// TIA Portal V17 export
// export: Created 2025-07-01T14:26:13.4361158Z, ExportSetting WithDefaults, DisplayName Totally Integrated Automation Portal, DisplayVersion V17 Update 8, DisplayName TIA Portal Openness, DisplayVersion V17 Update 8, DisplayName TIA Portal Version Control Interface, DisplayVersion V17, DisplayName SINAMICS Startdrive Advanced, DisplayVersion V17 SP2, DisplayName SINAMICS Startdrive G110M, G120, G120C, G120D, G120P, G115D, DisplayVersion V17 SP2, DisplayName SINAMICS Startdrive G130, G150, S120, S150, SINAMICS MV, S210, DisplayVersion V17 SP2, DisplayName STEP 7 Professional, DisplayVersion V17 Update 8, DisplayName SINUMERIK ONE STEP 7 Toolbox, DisplayVersion V17 Update 12, DisplayName SINUMERIK ONE PLC Basic Program Plus, DisplayVersion V17 Update 12, DisplayName SINUMERIK 840D sl STEP 7 Toolbox, DisplayVersion V17 Update 12, DisplayName STEP 7 Safety, DisplayVersion V17 Update 6, DisplayName WinCC Advanced, DisplayVersion V17 Update 8
FUNCTION "FC17100_MAINTENANCE_HMI_SCREEN_VARIABLES" : Void   // FC17100, LAD
{ S7_Optimized_Access := 'TRUE' }
VERSION : 0.1
// stored: AutoNumber false, IsIECCheckEnabled false, SetENOAutomatically false, UDAEnableTagReadback false
   VAR_TEMP
      TEMP : Int;
      NUM_OF_HELPS_TO_0 : Int;
   END_VAR
BEGIN

REGION Network 1: ACTION DONE: POWDER > UNIT 1 > GENERAL
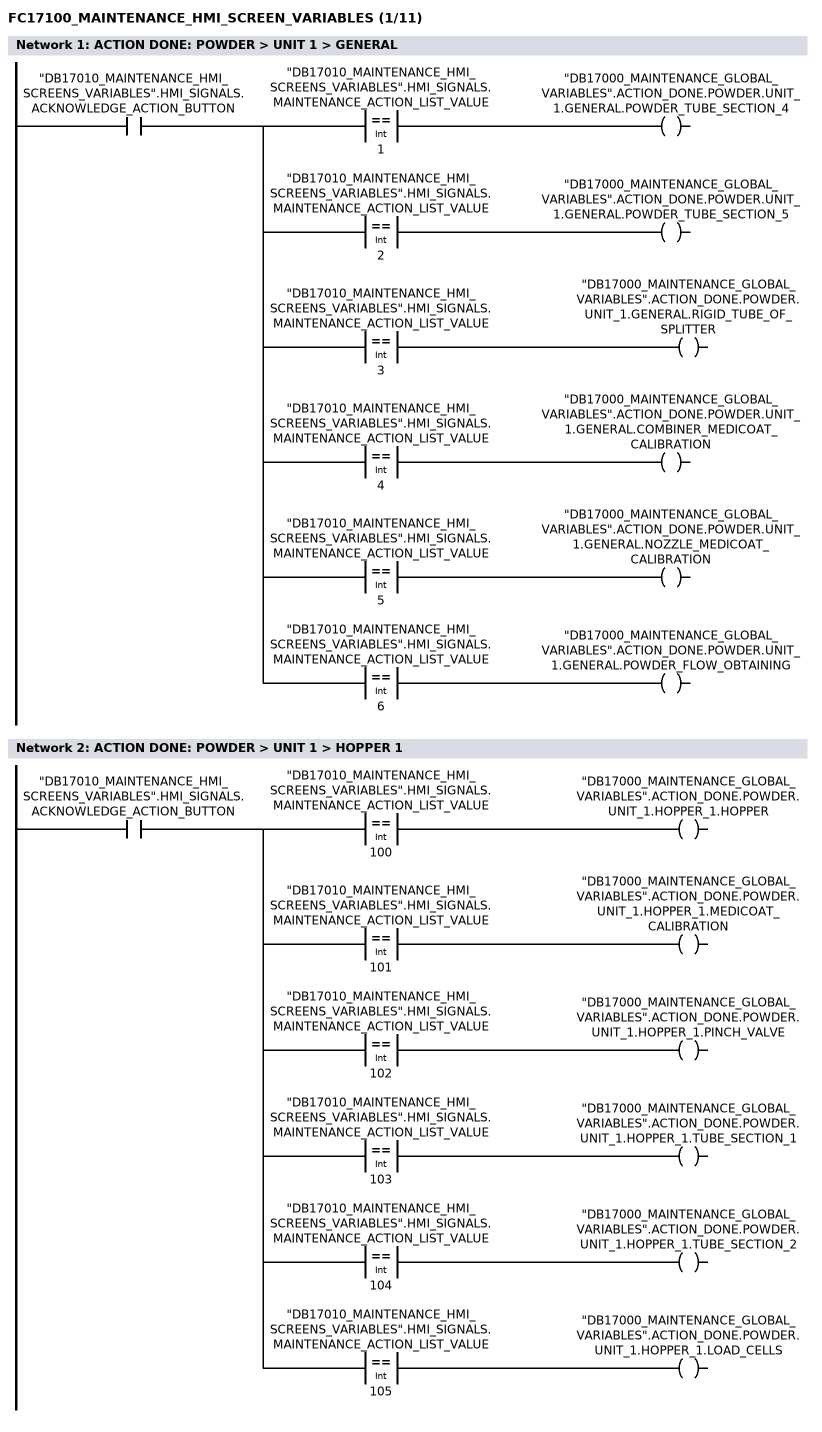
   RUNG wire#powerrail
      Contact( "DB17010_MAINTENANCE_HMI_SCREENS_VARIABLES".HMI_SIGNALS.ACKNOWLEDGE_ACTION_BUTTON )
      wire#w1
      { S7_Templates := "SrcType := Int" } EQ_Contact(in1 := "DB17010_MAINTENANCE_HMI_SCREENS_VARIABLES".HMI_SIGNALS.MAINTENANCE_ACTION_LIST_VALUE, in2 := 1)
      Coil( "DB17000_MAINTENANCE_GLOBAL_VARIABLES".ACTION_DONE.POWDER.UNIT_1.GENERAL.POWDER_TUBE_SECTION_4 )
   END_RUNG
   RUNG wire#w1
      { S7_Templates := "SrcType := Int" } EQ_Contact(in1 := "DB17010_MAINTENANCE_HMI_SCREENS_VARIABLES".HMI_SIGNALS.MAINTENANCE_ACTION_LIST_VALUE, in2 := 2)
      Coil( "DB17000_MAINTENANCE_GLOBAL_VARIABLES".ACTION_DONE.POWDER.UNIT_1.GENERAL.POWDER_TUBE_SECTION_5 )
   END_RUNG
   RUNG wire#w1
      { S7_Templates := "SrcType := Int" } EQ_Contact(in1 := "DB17010_MAINTENANCE_HMI_SCREENS_VARIABLES".HMI_SIGNALS.MAINTENANCE_ACTION_LIST_VALUE, in2 := 3)
      Coil( "DB17000_MAINTENANCE_GLOBAL_VARIABLES".ACTION_DONE.POWDER.UNIT_1.GENERAL.RIGID_TUBE_OF_SPLITTER )
   END_RUNG
   RUNG wire#w1
      { S7_Templates := "SrcType := Int" } EQ_Contact(in1 := "DB17010_MAINTENANCE_HMI_SCREENS_VARIABLES".HMI_SIGNALS.MAINTENANCE_ACTION_LIST_VALUE, in2 := 4)
      Coil( "DB17000_MAINTENANCE_GLOBAL_VARIABLES".ACTION_DONE.POWDER.UNIT_1.GENERAL.COMBINER_MEDICOAT_CALIBRATION )
   END_RUNG
   RUNG wire#w1
      { S7_Templates := "SrcType := Int" } EQ_Contact(in1 := "DB17010_MAINTENANCE_HMI_SCREENS_VARIABLES".HMI_SIGNALS.MAINTENANCE_ACTION_LIST_VALUE, in2 := 5)
      Coil( "DB17000_MAINTENANCE_GLOBAL_VARIABLES".ACTION_DONE.POWDER.UNIT_1.GENERAL.NOZZLE_MEDICOAT_CALIBRATION )
   END_RUNG
   RUNG wire#w1
      { S7_Templates := "SrcType := Int" } EQ_Contact(in1 := "DB17010_MAINTENANCE_HMI_SCREENS_VARIABLES".HMI_SIGNALS.MAINTENANCE_ACTION_LIST_VALUE, in2 := 6)
      Coil( "DB17000_MAINTENANCE_GLOBAL_VARIABLES".ACTION_DONE.POWDER.UNIT_1.GENERAL.POWDER_FLOW_OBTAINING )
   END_RUNG
   // the same network as SCL:
   "DB17000_MAINTENANCE_GLOBAL_VARIABLES".ACTION_DONE.POWDER.UNIT_1.GENERAL.POWDER_TUBE_SECTION_4 := "DB17010_MAINTENANCE_HMI_SCREENS_VARIABLES".HMI_SIGNALS.ACKNOWLEDGE_ACTION_BUTTON AND ("DB17010_MAINTENANCE_HMI_SCREENS_VARIABLES".HMI_SIGNALS.MAINTENANCE_ACTION_LIST_VALUE = 1);
   "DB17000_MAINTENANCE_GLOBAL_VARIABLES".ACTION_DONE.POWDER.UNIT_1.GENERAL.POWDER_TUBE_SECTION_5 := "DB17010_MAINTENANCE_HMI_SCREENS_VARIABLES".HMI_SIGNALS.ACKNOWLEDGE_ACTION_BUTTON AND ("DB17010_MAINTENANCE_HMI_SCREENS_VARIABLES".HMI_SIGNALS.MAINTENANCE_ACTION_LIST_VALUE = 2);
   "DB17000_MAINTENANCE_GLOBAL_VARIABLES".ACTION_DONE.POWDER.UNIT_1.GENERAL.RIGID_TUBE_OF_SPLITTER := "DB17010_MAINTENANCE_HMI_SCREENS_VARIABLES".HMI_SIGNALS.ACKNOWLEDGE_ACTION_BUTTON AND ("DB17010_MAINTENANCE_HMI_SCREENS_VARIABLES".HMI_SIGNALS.MAINTENANCE_ACTION_LIST_VALUE = 3);
   "DB17000_MAINTENANCE_GLOBAL_VARIABLES".ACTION_DONE.POWDER.UNIT_1.GENERAL.COMBINER_MEDICOAT_CALIBRATION := "DB17010_MAINTENANCE_HMI_SCREENS_VARIABLES".HMI_SIGNALS.ACKNOWLEDGE_ACTION_BUTTON AND ("DB17010_MAINTENANCE_HMI_SCREENS_VARIABLES".HMI_SIGNALS.MAINTENANCE_ACTION_LIST_VALUE = 4);
   "DB17000_MAINTENANCE_GLOBAL_VARIABLES".ACTION_DONE.POWDER.UNIT_1.GENERAL.NOZZLE_MEDICOAT_CALIBRATION := "DB17010_MAINTENANCE_HMI_SCREENS_VARIABLES".HMI_SIGNALS.ACKNOWLEDGE_ACTION_BUTTON AND ("DB17010_MAINTENANCE_HMI_SCREENS_VARIABLES".HMI_SIGNALS.MAINTENANCE_ACTION_LIST_VALUE = 5);
   "DB17000_MAINTENANCE_GLOBAL_VARIABLES".ACTION_DONE.POWDER.UNIT_1.GENERAL.POWDER_FLOW_OBTAINING := "DB17010_MAINTENANCE_HMI_SCREENS_VARIABLES".HMI_SIGNALS.ACKNOWLEDGE_ACTION_BUTTON AND ("DB17010_MAINTENANCE_HMI_SCREENS_VARIABLES".HMI_SIGNALS.MAINTENANCE_ACTION_LIST_VALUE = 6);
END_REGION

REGION Network 2: ACTION DONE: POWDER > UNIT 1 > HOPPER 1
   RUNG wire#powerrail
      Contact( "DB17010_MAINTENANCE_HMI_SCREENS_VARIABLES".HMI_SIGNALS.ACKNOWLEDGE_ACTION_BUTTON )
      wire#w1
      { S7_Templates := "SrcType := Int" } EQ_Contact(in1 := "DB17010_MAINTENANCE_HMI_SCREENS_VARIABLES".HMI_SIGNALS.MAINTENANCE_ACTION_LIST_VALUE, in2 := 100)
      Coil( "DB17000_MAINTENANCE_GLOBAL_VARIABLES".ACTION_DONE.POWDER.UNIT_1.HOPPER_1.HOPPER )
   END_RUNG
   RUNG wire#w1
      { S7_Templates := "SrcType := Int" } EQ_Contact(in1 := "DB17010_MAINTENANCE_HMI_SCREENS_VARIABLES".HMI_SIGNALS.MAINTENANCE_ACTION_LIST_VALUE, in2 := 101)
      Coil( "DB17000_MAINTENANCE_GLOBAL_VARIABLES".ACTION_DONE.POWDER.UNIT_1.HOPPER_1.MEDICOAT_CALIBRATION )
   END_RUNG
   RUNG wire#w1
      { S7_Templates := "SrcType := Int" } EQ_Contact(in1 := "DB17010_MAINTENANCE_HMI_SCREENS_VARIABLES".HMI_SIGNALS.MAINTENANCE_ACTION_LIST_VALUE, in2 := 102)
      Coil( "DB17000_MAINTENANCE_GLOBAL_VARIABLES".ACTION_DONE.POWDER.UNIT_1.HOPPER_1.PINCH_VALVE )
   END_RUNG
   RUNG wire#w1
      { S7_Templates := "SrcType := Int" } EQ_Contact(in1 := "DB17010_MAINTENANCE_HMI_SCREENS_VARIABLES".HMI_SIGNALS.MAINTENANCE_ACTION_LIST_VALUE, in2 := 103)
      Coil( "DB17000_MAINTENANCE_GLOBAL_VARIABLES".ACTION_DONE.POWDER.UNIT_1.HOPPER_1.TUBE_SECTION_1 )
   END_RUNG
   RUNG wire#w1
      { S7_Templates := "SrcType := Int" } EQ_Contact(in1 := "DB17010_MAINTENANCE_HMI_SCREENS_VARIABLES".HMI_SIGNALS.MAINTENANCE_ACTION_LIST_VALUE, in2 := 104)
      Coil( "DB17000_MAINTENANCE_GLOBAL_VARIABLES".ACTION_DONE.POWDER.UNIT_1.HOPPER_1.TUBE_SECTION_2 )
   END_RUNG
   RUNG wire#w1
      { S7_Templates := "SrcType := Int" } EQ_Contact(in1 := "DB17010_MAINTENANCE_HMI_SCREENS_VARIABLES".HMI_SIGNALS.MAINTENANCE_ACTION_LIST_VALUE, in2 := 105)
      Coil( "DB17000_MAINTENANCE_GLOBAL_VARIABLES".ACTION_DONE.POWDER.UNIT_1.HOPPER_1.LOAD_CELLS )
   END_RUNG
   // the same network as SCL:
   "DB17000_MAINTENANCE_GLOBAL_VARIABLES".ACTION_DONE.POWDER.UNIT_1.HOPPER_1.HOPPER := "DB17010_MAINTENANCE_HMI_SCREENS_VARIABLES".HMI_SIGNALS.ACKNOWLEDGE_ACTION_BUTTON AND ("DB17010_MAINTENANCE_HMI_SCREENS_VARIABLES".HMI_SIGNALS.MAINTENANCE_ACTION_LIST_VALUE = 100);
   "DB17000_MAINTENANCE_GLOBAL_VARIABLES".ACTION_DONE.POWDER.UNIT_1.HOPPER_1.MEDICOAT_CALIBRATION := "DB17010_MAINTENANCE_HMI_SCREENS_VARIABLES".HMI_SIGNALS.ACKNOWLEDGE_ACTION_BUTTON AND ("DB17010_MAINTENANCE_HMI_SCREENS_VARIABLES".HMI_SIGNALS.MAINTENANCE_ACTION_LIST_VALUE = 101);
   "DB17000_MAINTENANCE_GLOBAL_VARIABLES".ACTION_DONE.POWDER.UNIT_1.HOPPER_1.PINCH_VALVE := "DB17010_MAINTENANCE_HMI_SCREENS_VARIABLES".HMI_SIGNALS.ACKNOWLEDGE_ACTION_BUTTON AND ("DB17010_MAINTENANCE_HMI_SCREENS_VARIABLES".HMI_SIGNALS.MAINTENANCE_ACTION_LIST_VALUE = 102);
   "DB17000_MAINTENANCE_GLOBAL_VARIABLES".ACTION_DONE.POWDER.UNIT_1.HOPPER_1.TUBE_SECTION_1 := "DB17010_MAINTENANCE_HMI_SCREENS_VARIABLES".HMI_SIGNALS.ACKNOWLEDGE_ACTION_BUTTON AND ("DB17010_MAINTENANCE_HMI_SCREENS_VARIABLES".HMI_SIGNALS.MAINTENANCE_ACTION_LIST_VALUE = 103);
   "DB17000_MAINTENANCE_GLOBAL_VARIABLES".ACTION_DONE.POWDER.UNIT_1.HOPPER_1.TUBE_SECTION_2 := "DB17010_MAINTENANCE_HMI_SCREENS_VARIABLES".HMI_SIGNALS.ACKNOWLEDGE_ACTION_BUTTON AND ("DB17010_MAINTENANCE_HMI_SCREENS_VARIABLES".HMI_SIGNALS.MAINTENANCE_ACTION_LIST_VALUE = 104);
   "DB17000_MAINTENANCE_GLOBAL_VARIABLES".ACTION_DONE.POWDER.UNIT_1.HOPPER_1.LOAD_CELLS := "DB17010_MAINTENANCE_HMI_SCREENS_VARIABLES".HMI_SIGNALS.ACKNOWLEDGE_ACTION_BUTTON AND ("DB17010_MAINTENANCE_HMI_SCREENS_VARIABLES".HMI_SIGNALS.MAINTENANCE_ACTION_LIST_VALUE = 105);
END_REGION

REGION Network 3: ACTION DONE: POWDER > UNIT 1 > HOPPER 2
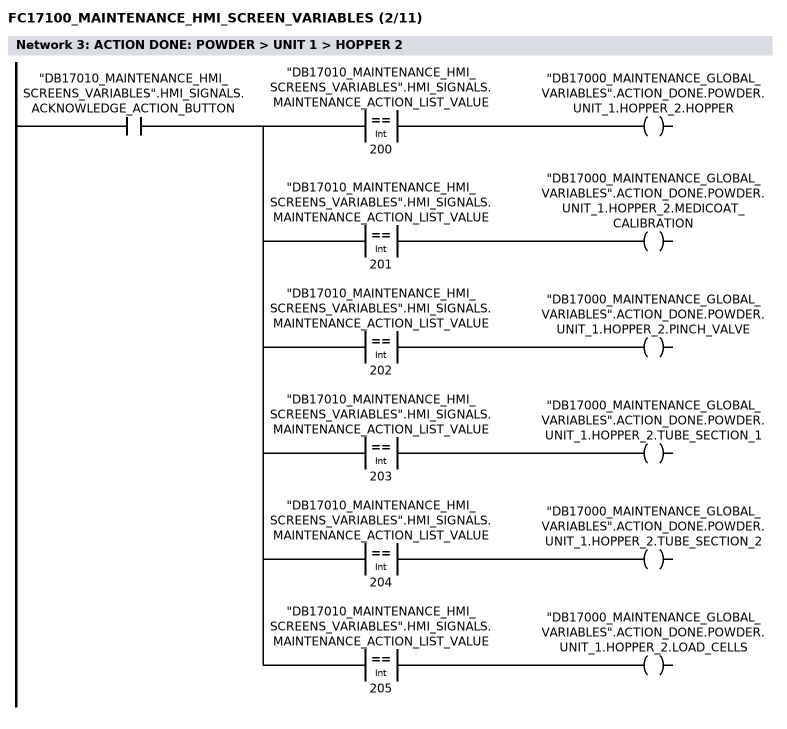
   RUNG wire#powerrail
      Contact( "DB17010_MAINTENANCE_HMI_SCREENS_VARIABLES".HMI_SIGNALS.ACKNOWLEDGE_ACTION_BUTTON )
      wire#w1
      { S7_Templates := "SrcType := Int" } EQ_Contact(in1 := "DB17010_MAINTENANCE_HMI_SCREENS_VARIABLES".HMI_SIGNALS.MAINTENANCE_ACTION_LIST_VALUE, in2 := 200)
      Coil( "DB17000_MAINTENANCE_GLOBAL_VARIABLES".ACTION_DONE.POWDER.UNIT_1.HOPPER_2.HOPPER )
   END_RUNG
   RUNG wire#w1
      { S7_Templates := "SrcType := Int" } EQ_Contact(in1 := "DB17010_MAINTENANCE_HMI_SCREENS_VARIABLES".HMI_SIGNALS.MAINTENANCE_ACTION_LIST_VALUE, in2 := 201)
      Coil( "DB17000_MAINTENANCE_GLOBAL_VARIABLES".ACTION_DONE.POWDER.UNIT_1.HOPPER_2.MEDICOAT_CALIBRATION )
   END_RUNG
   RUNG wire#w1
      { S7_Templates := "SrcType := Int" } EQ_Contact(in1 := "DB17010_MAINTENANCE_HMI_SCREENS_VARIABLES".HMI_SIGNALS.MAINTENANCE_ACTION_LIST_VALUE, in2 := 202)
      Coil( "DB17000_MAINTENANCE_GLOBAL_VARIABLES".ACTION_DONE.POWDER.UNIT_1.HOPPER_2.PINCH_VALVE )
   END_RUNG
   RUNG wire#w1
      { S7_Templates := "SrcType := Int" } EQ_Contact(in1 := "DB17010_MAINTENANCE_HMI_SCREENS_VARIABLES".HMI_SIGNALS.MAINTENANCE_ACTION_LIST_VALUE, in2 := 203)
      Coil( "DB17000_MAINTENANCE_GLOBAL_VARIABLES".ACTION_DONE.POWDER.UNIT_1.HOPPER_2.TUBE_SECTION_1 )
   END_RUNG
   RUNG wire#w1
      { S7_Templates := "SrcType := Int" } EQ_Contact(in1 := "DB17010_MAINTENANCE_HMI_SCREENS_VARIABLES".HMI_SIGNALS.MAINTENANCE_ACTION_LIST_VALUE, in2 := 204)
      Coil( "DB17000_MAINTENANCE_GLOBAL_VARIABLES".ACTION_DONE.POWDER.UNIT_1.HOPPER_2.TUBE_SECTION_2 )
   END_RUNG
   RUNG wire#w1
      { S7_Templates := "SrcType := Int" } EQ_Contact(in1 := "DB17010_MAINTENANCE_HMI_SCREENS_VARIABLES".HMI_SIGNALS.MAINTENANCE_ACTION_LIST_VALUE, in2 := 205)
      Coil( "DB17000_MAINTENANCE_GLOBAL_VARIABLES".ACTION_DONE.POWDER.UNIT_1.HOPPER_2.LOAD_CELLS )
   END_RUNG
   // the same network as SCL:
   "DB17000_MAINTENANCE_GLOBAL_VARIABLES".ACTION_DONE.POWDER.UNIT_1.HOPPER_2.HOPPER := "DB17010_MAINTENANCE_HMI_SCREENS_VARIABLES".HMI_SIGNALS.ACKNOWLEDGE_ACTION_BUTTON AND ("DB17010_MAINTENANCE_HMI_SCREENS_VARIABLES".HMI_SIGNALS.MAINTENANCE_ACTION_LIST_VALUE = 200);
   "DB17000_MAINTENANCE_GLOBAL_VARIABLES".ACTION_DONE.POWDER.UNIT_1.HOPPER_2.MEDICOAT_CALIBRATION := "DB17010_MAINTENANCE_HMI_SCREENS_VARIABLES".HMI_SIGNALS.ACKNOWLEDGE_ACTION_BUTTON AND ("DB17010_MAINTENANCE_HMI_SCREENS_VARIABLES".HMI_SIGNALS.MAINTENANCE_ACTION_LIST_VALUE = 201);
   "DB17000_MAINTENANCE_GLOBAL_VARIABLES".ACTION_DONE.POWDER.UNIT_1.HOPPER_2.PINCH_VALVE := "DB17010_MAINTENANCE_HMI_SCREENS_VARIABLES".HMI_SIGNALS.ACKNOWLEDGE_ACTION_BUTTON AND ("DB17010_MAINTENANCE_HMI_SCREENS_VARIABLES".HMI_SIGNALS.MAINTENANCE_ACTION_LIST_VALUE = 202);
   "DB17000_MAINTENANCE_GLOBAL_VARIABLES".ACTION_DONE.POWDER.UNIT_1.HOPPER_2.TUBE_SECTION_1 := "DB17010_MAINTENANCE_HMI_SCREENS_VARIABLES".HMI_SIGNALS.ACKNOWLEDGE_ACTION_BUTTON AND ("DB17010_MAINTENANCE_HMI_SCREENS_VARIABLES".HMI_SIGNALS.MAINTENANCE_ACTION_LIST_VALUE = 203);
   "DB17000_MAINTENANCE_GLOBAL_VARIABLES".ACTION_DONE.POWDER.UNIT_1.HOPPER_2.TUBE_SECTION_2 := "DB17010_MAINTENANCE_HMI_SCREENS_VARIABLES".HMI_SIGNALS.ACKNOWLEDGE_ACTION_BUTTON AND ("DB17010_MAINTENANCE_HMI_SCREENS_VARIABLES".HMI_SIGNALS.MAINTENANCE_ACTION_LIST_VALUE = 204);
   "DB17000_MAINTENANCE_GLOBAL_VARIABLES".ACTION_DONE.POWDER.UNIT_1.HOPPER_2.LOAD_CELLS := "DB17010_MAINTENANCE_HMI_SCREENS_VARIABLES".HMI_SIGNALS.ACKNOWLEDGE_ACTION_BUTTON AND ("DB17010_MAINTENANCE_HMI_SCREENS_VARIABLES".HMI_SIGNALS.MAINTENANCE_ACTION_LIST_VALUE = 205);
END_REGION

REGION Network 4: ACTION DONE: POWDER > UNIT 1 > FEEDER 1
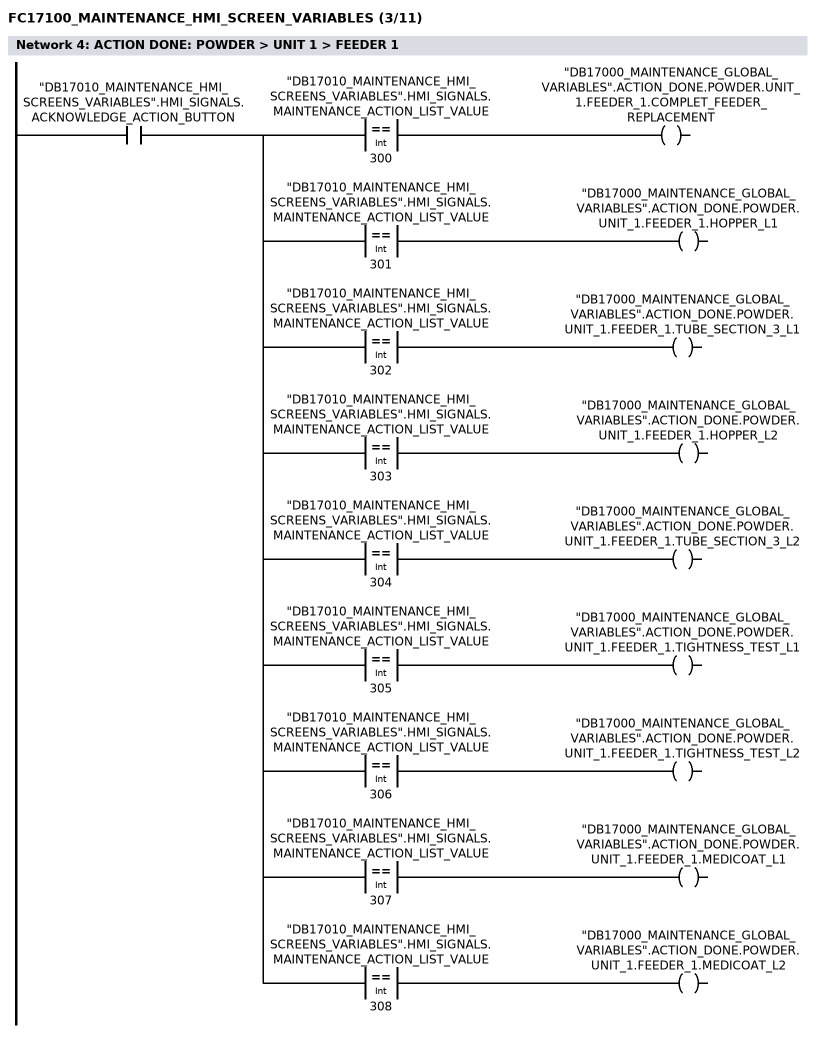
   RUNG wire#powerrail
      Contact( "DB17010_MAINTENANCE_HMI_SCREENS_VARIABLES".HMI_SIGNALS.ACKNOWLEDGE_ACTION_BUTTON )
      wire#w1
      { S7_Templates := "SrcType := Int" } EQ_Contact(in1 := "DB17010_MAINTENANCE_HMI_SCREENS_VARIABLES".HMI_SIGNALS.MAINTENANCE_ACTION_LIST_VALUE, in2 := 300)
      Coil( "DB17000_MAINTENANCE_GLOBAL_VARIABLES".ACTION_DONE.POWDER.UNIT_1.FEEDER_1.COMPLET_FEEDER_REPLACEMENT )
   END_RUNG
   RUNG wire#w1
      { S7_Templates := "SrcType := Int" } EQ_Contact(in1 := "DB17010_MAINTENANCE_HMI_SCREENS_VARIABLES".HMI_SIGNALS.MAINTENANCE_ACTION_LIST_VALUE, in2 := 301)
      Coil( "DB17000_MAINTENANCE_GLOBAL_VARIABLES".ACTION_DONE.POWDER.UNIT_1.FEEDER_1.HOPPER_L1 )
   END_RUNG
   RUNG wire#w1
      { S7_Templates := "SrcType := Int" } EQ_Contact(in1 := "DB17010_MAINTENANCE_HMI_SCREENS_VARIABLES".HMI_SIGNALS.MAINTENANCE_ACTION_LIST_VALUE, in2 := 302)
      Coil( "DB17000_MAINTENANCE_GLOBAL_VARIABLES".ACTION_DONE.POWDER.UNIT_1.FEEDER_1.TUBE_SECTION_3_L1 )
   END_RUNG
   RUNG wire#w1
      { S7_Templates := "SrcType := Int" } EQ_Contact(in1 := "DB17010_MAINTENANCE_HMI_SCREENS_VARIABLES".HMI_SIGNALS.MAINTENANCE_ACTION_LIST_VALUE, in2 := 303)
      Coil( "DB17000_MAINTENANCE_GLOBAL_VARIABLES".ACTION_DONE.POWDER.UNIT_1.FEEDER_1.HOPPER_L2 )
   END_RUNG
   RUNG wire#w1
      { S7_Templates := "SrcType := Int" } EQ_Contact(in1 := "DB17010_MAINTENANCE_HMI_SCREENS_VARIABLES".HMI_SIGNALS.MAINTENANCE_ACTION_LIST_VALUE, in2 := 304)
      Coil( "DB17000_MAINTENANCE_GLOBAL_VARIABLES".ACTION_DONE.POWDER.UNIT_1.FEEDER_1.TUBE_SECTION_3_L2 )
   END_RUNG
   RUNG wire#w1
      { S7_Templates := "SrcType := Int" } EQ_Contact(in1 := "DB17010_MAINTENANCE_HMI_SCREENS_VARIABLES".HMI_SIGNALS.MAINTENANCE_ACTION_LIST_VALUE, in2 := 305)
      Coil( "DB17000_MAINTENANCE_GLOBAL_VARIABLES".ACTION_DONE.POWDER.UNIT_1.FEEDER_1.TIGHTNESS_TEST_L1 )
   END_RUNG
   RUNG wire#w1
      { S7_Templates := "SrcType := Int" } EQ_Contact(in1 := "DB17010_MAINTENANCE_HMI_SCREENS_VARIABLES".HMI_SIGNALS.MAINTENANCE_ACTION_LIST_VALUE, in2 := 306)
      Coil( "DB17000_MAINTENANCE_GLOBAL_VARIABLES".ACTION_DONE.POWDER.UNIT_1.FEEDER_1.TIGHTNESS_TEST_L2 )
   END_RUNG
   RUNG wire#w1
      { S7_Templates := "SrcType := Int" } EQ_Contact(in1 := "DB17010_MAINTENANCE_HMI_SCREENS_VARIABLES".HMI_SIGNALS.MAINTENANCE_ACTION_LIST_VALUE, in2 := 307)
      Coil( "DB17000_MAINTENANCE_GLOBAL_VARIABLES".ACTION_DONE.POWDER.UNIT_1.FEEDER_1.MEDICOAT_L1 )
   END_RUNG
   RUNG wire#w1
      { S7_Templates := "SrcType := Int" } EQ_Contact(in1 := "DB17010_MAINTENANCE_HMI_SCREENS_VARIABLES".HMI_SIGNALS.MAINTENANCE_ACTION_LIST_VALUE, in2 := 308)
      Coil( "DB17000_MAINTENANCE_GLOBAL_VARIABLES".ACTION_DONE.POWDER.UNIT_1.FEEDER_1.MEDICOAT_L2 )
   END_RUNG
   // the same network as SCL:
   "DB17000_MAINTENANCE_GLOBAL_VARIABLES".ACTION_DONE.POWDER.UNIT_1.FEEDER_1.COMPLET_FEEDER_REPLACEMENT := "DB17010_MAINTENANCE_HMI_SCREENS_VARIABLES".HMI_SIGNALS.ACKNOWLEDGE_ACTION_BUTTON AND ("DB17010_MAINTENANCE_HMI_SCREENS_VARIABLES".HMI_SIGNALS.MAINTENANCE_ACTION_LIST_VALUE = 300);
   "DB17000_MAINTENANCE_GLOBAL_VARIABLES".ACTION_DONE.POWDER.UNIT_1.FEEDER_1.HOPPER_L1 := "DB17010_MAINTENANCE_HMI_SCREENS_VARIABLES".HMI_SIGNALS.ACKNOWLEDGE_ACTION_BUTTON AND ("DB17010_MAINTENANCE_HMI_SCREENS_VARIABLES".HMI_SIGNALS.MAINTENANCE_ACTION_LIST_VALUE = 301);
   "DB17000_MAINTENANCE_GLOBAL_VARIABLES".ACTION_DONE.POWDER.UNIT_1.FEEDER_1.TUBE_SECTION_3_L1 := "DB17010_MAINTENANCE_HMI_SCREENS_VARIABLES".HMI_SIGNALS.ACKNOWLEDGE_ACTION_BUTTON AND ("DB17010_MAINTENANCE_HMI_SCREENS_VARIABLES".HMI_SIGNALS.MAINTENANCE_ACTION_LIST_VALUE = 302);
   "DB17000_MAINTENANCE_GLOBAL_VARIABLES".ACTION_DONE.POWDER.UNIT_1.FEEDER_1.HOPPER_L2 := "DB17010_MAINTENANCE_HMI_SCREENS_VARIABLES".HMI_SIGNALS.ACKNOWLEDGE_ACTION_BUTTON AND ("DB17010_MAINTENANCE_HMI_SCREENS_VARIABLES".HMI_SIGNALS.MAINTENANCE_ACTION_LIST_VALUE = 303);
   "DB17000_MAINTENANCE_GLOBAL_VARIABLES".ACTION_DONE.POWDER.UNIT_1.FEEDER_1.TUBE_SECTION_3_L2 := "DB17010_MAINTENANCE_HMI_SCREENS_VARIABLES".HMI_SIGNALS.ACKNOWLEDGE_ACTION_BUTTON AND ("DB17010_MAINTENANCE_HMI_SCREENS_VARIABLES".HMI_SIGNALS.MAINTENANCE_ACTION_LIST_VALUE = 304);
   "DB17000_MAINTENANCE_GLOBAL_VARIABLES".ACTION_DONE.POWDER.UNIT_1.FEEDER_1.TIGHTNESS_TEST_L1 := "DB17010_MAINTENANCE_HMI_SCREENS_VARIABLES".HMI_SIGNALS.ACKNOWLEDGE_ACTION_BUTTON AND ("DB17010_MAINTENANCE_HMI_SCREENS_VARIABLES".HMI_SIGNALS.MAINTENANCE_ACTION_LIST_VALUE = 305);
   "DB17000_MAINTENANCE_GLOBAL_VARIABLES".ACTION_DONE.POWDER.UNIT_1.FEEDER_1.TIGHTNESS_TEST_L2 := "DB17010_MAINTENANCE_HMI_SCREENS_VARIABLES".HMI_SIGNALS.ACKNOWLEDGE_ACTION_BUTTON AND ("DB17010_MAINTENANCE_HMI_SCREENS_VARIABLES".HMI_SIGNALS.MAINTENANCE_ACTION_LIST_VALUE = 306);
   "DB17000_MAINTENANCE_GLOBAL_VARIABLES".ACTION_DONE.POWDER.UNIT_1.FEEDER_1.MEDICOAT_L1 := "DB17010_MAINTENANCE_HMI_SCREENS_VARIABLES".HMI_SIGNALS.ACKNOWLEDGE_ACTION_BUTTON AND ("DB17010_MAINTENANCE_HMI_SCREENS_VARIABLES".HMI_SIGNALS.MAINTENANCE_ACTION_LIST_VALUE = 307);
   "DB17000_MAINTENANCE_GLOBAL_VARIABLES".ACTION_DONE.POWDER.UNIT_1.FEEDER_1.MEDICOAT_L2 := "DB17010_MAINTENANCE_HMI_SCREENS_VARIABLES".HMI_SIGNALS.ACKNOWLEDGE_ACTION_BUTTON AND ("DB17010_MAINTENANCE_HMI_SCREENS_VARIABLES".HMI_SIGNALS.MAINTENANCE_ACTION_LIST_VALUE = 308);
END_REGION

REGION Network 5: ACTION DONE: POWDER > UNIT 2 > GENERAL
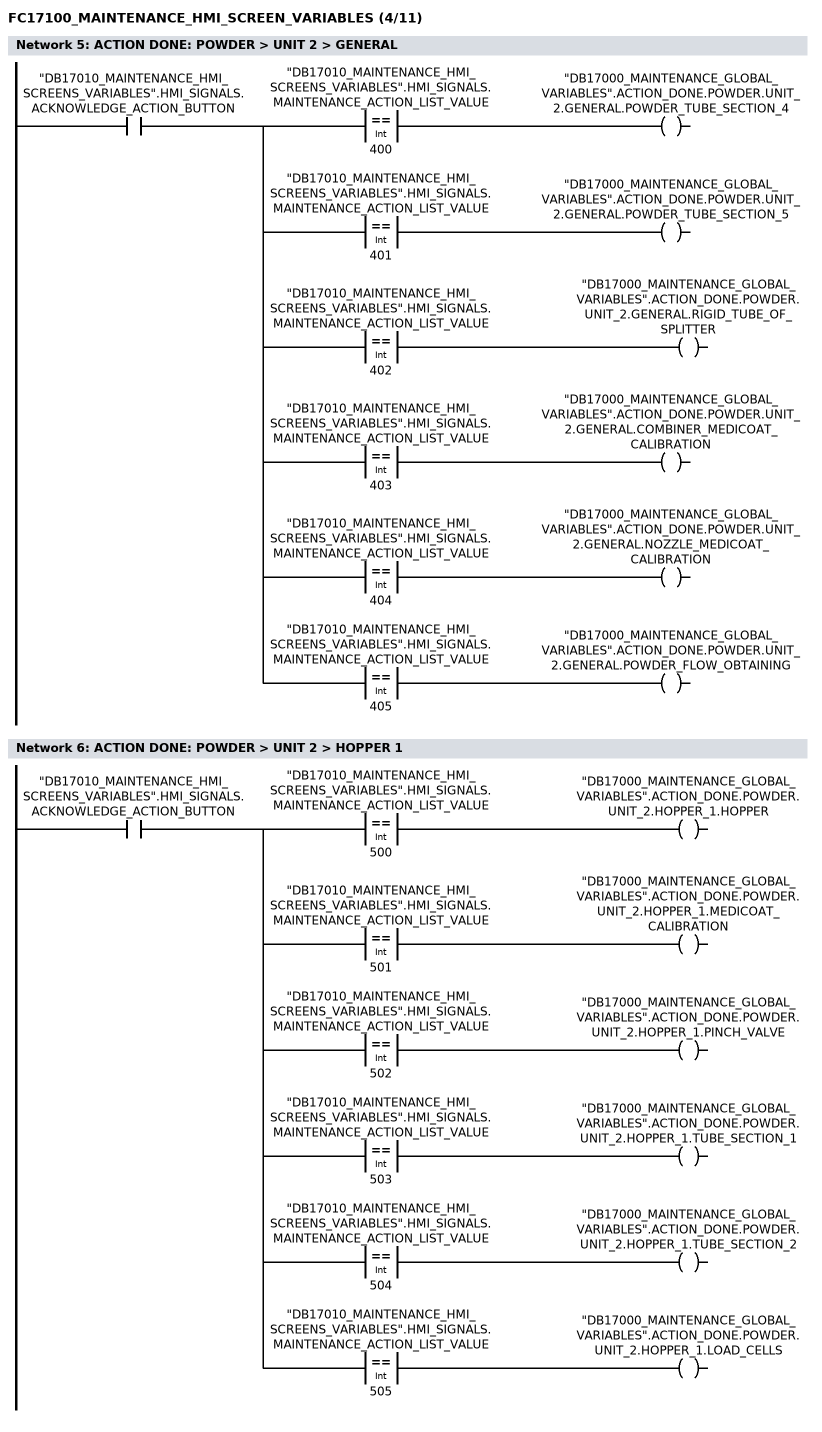
   RUNG wire#powerrail
      Contact( "DB17010_MAINTENANCE_HMI_SCREENS_VARIABLES".HMI_SIGNALS.ACKNOWLEDGE_ACTION_BUTTON )
      wire#w1
      { S7_Templates := "SrcType := Int" } EQ_Contact(in1 := "DB17010_MAINTENANCE_HMI_SCREENS_VARIABLES".HMI_SIGNALS.MAINTENANCE_ACTION_LIST_VALUE, in2 := 400)
      Coil( "DB17000_MAINTENANCE_GLOBAL_VARIABLES".ACTION_DONE.POWDER.UNIT_2.GENERAL.POWDER_TUBE_SECTION_4 )
   END_RUNG
   RUNG wire#w1
      { S7_Templates := "SrcType := Int" } EQ_Contact(in1 := "DB17010_MAINTENANCE_HMI_SCREENS_VARIABLES".HMI_SIGNALS.MAINTENANCE_ACTION_LIST_VALUE, in2 := 401)
      Coil( "DB17000_MAINTENANCE_GLOBAL_VARIABLES".ACTION_DONE.POWDER.UNIT_2.GENERAL.POWDER_TUBE_SECTION_5 )
   END_RUNG
   RUNG wire#w1
      { S7_Templates := "SrcType := Int" } EQ_Contact(in1 := "DB17010_MAINTENANCE_HMI_SCREENS_VARIABLES".HMI_SIGNALS.MAINTENANCE_ACTION_LIST_VALUE, in2 := 402)
      Coil( "DB17000_MAINTENANCE_GLOBAL_VARIABLES".ACTION_DONE.POWDER.UNIT_2.GENERAL.RIGID_TUBE_OF_SPLITTER )
   END_RUNG
   RUNG wire#w1
      { S7_Templates := "SrcType := Int" } EQ_Contact(in1 := "DB17010_MAINTENANCE_HMI_SCREENS_VARIABLES".HMI_SIGNALS.MAINTENANCE_ACTION_LIST_VALUE, in2 := 403)
      Coil( "DB17000_MAINTENANCE_GLOBAL_VARIABLES".ACTION_DONE.POWDER.UNIT_2.GENERAL.COMBINER_MEDICOAT_CALIBRATION )
   END_RUNG
   RUNG wire#w1
      { S7_Templates := "SrcType := Int" } EQ_Contact(in1 := "DB17010_MAINTENANCE_HMI_SCREENS_VARIABLES".HMI_SIGNALS.MAINTENANCE_ACTION_LIST_VALUE, in2 := 404)
      Coil( "DB17000_MAINTENANCE_GLOBAL_VARIABLES".ACTION_DONE.POWDER.UNIT_2.GENERAL.NOZZLE_MEDICOAT_CALIBRATION )
   END_RUNG
   RUNG wire#w1
      { S7_Templates := "SrcType := Int" } EQ_Contact(in1 := "DB17010_MAINTENANCE_HMI_SCREENS_VARIABLES".HMI_SIGNALS.MAINTENANCE_ACTION_LIST_VALUE, in2 := 405)
      Coil( "DB17000_MAINTENANCE_GLOBAL_VARIABLES".ACTION_DONE.POWDER.UNIT_2.GENERAL.POWDER_FLOW_OBTAINING )
   END_RUNG
   // the same network as SCL:
   "DB17000_MAINTENANCE_GLOBAL_VARIABLES".ACTION_DONE.POWDER.UNIT_2.GENERAL.POWDER_TUBE_SECTION_4 := "DB17010_MAINTENANCE_HMI_SCREENS_VARIABLES".HMI_SIGNALS.ACKNOWLEDGE_ACTION_BUTTON AND ("DB17010_MAINTENANCE_HMI_SCREENS_VARIABLES".HMI_SIGNALS.MAINTENANCE_ACTION_LIST_VALUE = 400);
   "DB17000_MAINTENANCE_GLOBAL_VARIABLES".ACTION_DONE.POWDER.UNIT_2.GENERAL.POWDER_TUBE_SECTION_5 := "DB17010_MAINTENANCE_HMI_SCREENS_VARIABLES".HMI_SIGNALS.ACKNOWLEDGE_ACTION_BUTTON AND ("DB17010_MAINTENANCE_HMI_SCREENS_VARIABLES".HMI_SIGNALS.MAINTENANCE_ACTION_LIST_VALUE = 401);
   "DB17000_MAINTENANCE_GLOBAL_VARIABLES".ACTION_DONE.POWDER.UNIT_2.GENERAL.RIGID_TUBE_OF_SPLITTER := "DB17010_MAINTENANCE_HMI_SCREENS_VARIABLES".HMI_SIGNALS.ACKNOWLEDGE_ACTION_BUTTON AND ("DB17010_MAINTENANCE_HMI_SCREENS_VARIABLES".HMI_SIGNALS.MAINTENANCE_ACTION_LIST_VALUE = 402);
   "DB17000_MAINTENANCE_GLOBAL_VARIABLES".ACTION_DONE.POWDER.UNIT_2.GENERAL.COMBINER_MEDICOAT_CALIBRATION := "DB17010_MAINTENANCE_HMI_SCREENS_VARIABLES".HMI_SIGNALS.ACKNOWLEDGE_ACTION_BUTTON AND ("DB17010_MAINTENANCE_HMI_SCREENS_VARIABLES".HMI_SIGNALS.MAINTENANCE_ACTION_LIST_VALUE = 403);
   "DB17000_MAINTENANCE_GLOBAL_VARIABLES".ACTION_DONE.POWDER.UNIT_2.GENERAL.NOZZLE_MEDICOAT_CALIBRATION := "DB17010_MAINTENANCE_HMI_SCREENS_VARIABLES".HMI_SIGNALS.ACKNOWLEDGE_ACTION_BUTTON AND ("DB17010_MAINTENANCE_HMI_SCREENS_VARIABLES".HMI_SIGNALS.MAINTENANCE_ACTION_LIST_VALUE = 404);
   "DB17000_MAINTENANCE_GLOBAL_VARIABLES".ACTION_DONE.POWDER.UNIT_2.GENERAL.POWDER_FLOW_OBTAINING := "DB17010_MAINTENANCE_HMI_SCREENS_VARIABLES".HMI_SIGNALS.ACKNOWLEDGE_ACTION_BUTTON AND ("DB17010_MAINTENANCE_HMI_SCREENS_VARIABLES".HMI_SIGNALS.MAINTENANCE_ACTION_LIST_VALUE = 405);
END_REGION

REGION Network 6: ACTION DONE: POWDER > UNIT 2 > HOPPER 1
   RUNG wire#powerrail
      Contact( "DB17010_MAINTENANCE_HMI_SCREENS_VARIABLES".HMI_SIGNALS.ACKNOWLEDGE_ACTION_BUTTON )
      wire#w1
      { S7_Templates := "SrcType := Int" } EQ_Contact(in1 := "DB17010_MAINTENANCE_HMI_SCREENS_VARIABLES".HMI_SIGNALS.MAINTENANCE_ACTION_LIST_VALUE, in2 := 500)
      Coil( "DB17000_MAINTENANCE_GLOBAL_VARIABLES".ACTION_DONE.POWDER.UNIT_2.HOPPER_1.HOPPER )
   END_RUNG
   RUNG wire#w1
      { S7_Templates := "SrcType := Int" } EQ_Contact(in1 := "DB17010_MAINTENANCE_HMI_SCREENS_VARIABLES".HMI_SIGNALS.MAINTENANCE_ACTION_LIST_VALUE, in2 := 501)
      Coil( "DB17000_MAINTENANCE_GLOBAL_VARIABLES".ACTION_DONE.POWDER.UNIT_2.HOPPER_1.MEDICOAT_CALIBRATION )
   END_RUNG
   RUNG wire#w1
      { S7_Templates := "SrcType := Int" } EQ_Contact(in1 := "DB17010_MAINTENANCE_HMI_SCREENS_VARIABLES".HMI_SIGNALS.MAINTENANCE_ACTION_LIST_VALUE, in2 := 502)
      Coil( "DB17000_MAINTENANCE_GLOBAL_VARIABLES".ACTION_DONE.POWDER.UNIT_2.HOPPER_1.PINCH_VALVE )
   END_RUNG
   RUNG wire#w1
      { S7_Templates := "SrcType := Int" } EQ_Contact(in1 := "DB17010_MAINTENANCE_HMI_SCREENS_VARIABLES".HMI_SIGNALS.MAINTENANCE_ACTION_LIST_VALUE, in2 := 503)
      Coil( "DB17000_MAINTENANCE_GLOBAL_VARIABLES".ACTION_DONE.POWDER.UNIT_2.HOPPER_1.TUBE_SECTION_1 )
   END_RUNG
   RUNG wire#w1
      { S7_Templates := "SrcType := Int" } EQ_Contact(in1 := "DB17010_MAINTENANCE_HMI_SCREENS_VARIABLES".HMI_SIGNALS.MAINTENANCE_ACTION_LIST_VALUE, in2 := 504)
      Coil( "DB17000_MAINTENANCE_GLOBAL_VARIABLES".ACTION_DONE.POWDER.UNIT_2.HOPPER_1.TUBE_SECTION_2 )
   END_RUNG
   RUNG wire#w1
      { S7_Templates := "SrcType := Int" } EQ_Contact(in1 := "DB17010_MAINTENANCE_HMI_SCREENS_VARIABLES".HMI_SIGNALS.MAINTENANCE_ACTION_LIST_VALUE, in2 := 505)
      Coil( "DB17000_MAINTENANCE_GLOBAL_VARIABLES".ACTION_DONE.POWDER.UNIT_2.HOPPER_1.LOAD_CELLS )
   END_RUNG
   // the same network as SCL:
   "DB17000_MAINTENANCE_GLOBAL_VARIABLES".ACTION_DONE.POWDER.UNIT_2.HOPPER_1.HOPPER := "DB17010_MAINTENANCE_HMI_SCREENS_VARIABLES".HMI_SIGNALS.ACKNOWLEDGE_ACTION_BUTTON AND ("DB17010_MAINTENANCE_HMI_SCREENS_VARIABLES".HMI_SIGNALS.MAINTENANCE_ACTION_LIST_VALUE = 500);
   "DB17000_MAINTENANCE_GLOBAL_VARIABLES".ACTION_DONE.POWDER.UNIT_2.HOPPER_1.MEDICOAT_CALIBRATION := "DB17010_MAINTENANCE_HMI_SCREENS_VARIABLES".HMI_SIGNALS.ACKNOWLEDGE_ACTION_BUTTON AND ("DB17010_MAINTENANCE_HMI_SCREENS_VARIABLES".HMI_SIGNALS.MAINTENANCE_ACTION_LIST_VALUE = 501);
   "DB17000_MAINTENANCE_GLOBAL_VARIABLES".ACTION_DONE.POWDER.UNIT_2.HOPPER_1.PINCH_VALVE := "DB17010_MAINTENANCE_HMI_SCREENS_VARIABLES".HMI_SIGNALS.ACKNOWLEDGE_ACTION_BUTTON AND ("DB17010_MAINTENANCE_HMI_SCREENS_VARIABLES".HMI_SIGNALS.MAINTENANCE_ACTION_LIST_VALUE = 502);
   "DB17000_MAINTENANCE_GLOBAL_VARIABLES".ACTION_DONE.POWDER.UNIT_2.HOPPER_1.TUBE_SECTION_1 := "DB17010_MAINTENANCE_HMI_SCREENS_VARIABLES".HMI_SIGNALS.ACKNOWLEDGE_ACTION_BUTTON AND ("DB17010_MAINTENANCE_HMI_SCREENS_VARIABLES".HMI_SIGNALS.MAINTENANCE_ACTION_LIST_VALUE = 503);
   "DB17000_MAINTENANCE_GLOBAL_VARIABLES".ACTION_DONE.POWDER.UNIT_2.HOPPER_1.TUBE_SECTION_2 := "DB17010_MAINTENANCE_HMI_SCREENS_VARIABLES".HMI_SIGNALS.ACKNOWLEDGE_ACTION_BUTTON AND ("DB17010_MAINTENANCE_HMI_SCREENS_VARIABLES".HMI_SIGNALS.MAINTENANCE_ACTION_LIST_VALUE = 504);
   "DB17000_MAINTENANCE_GLOBAL_VARIABLES".ACTION_DONE.POWDER.UNIT_2.HOPPER_1.LOAD_CELLS := "DB17010_MAINTENANCE_HMI_SCREENS_VARIABLES".HMI_SIGNALS.ACKNOWLEDGE_ACTION_BUTTON AND ("DB17010_MAINTENANCE_HMI_SCREENS_VARIABLES".HMI_SIGNALS.MAINTENANCE_ACTION_LIST_VALUE = 505);
END_REGION

REGION Network 7: ACTION DONE: POWDER > UNIT 2 > HOPPER 2
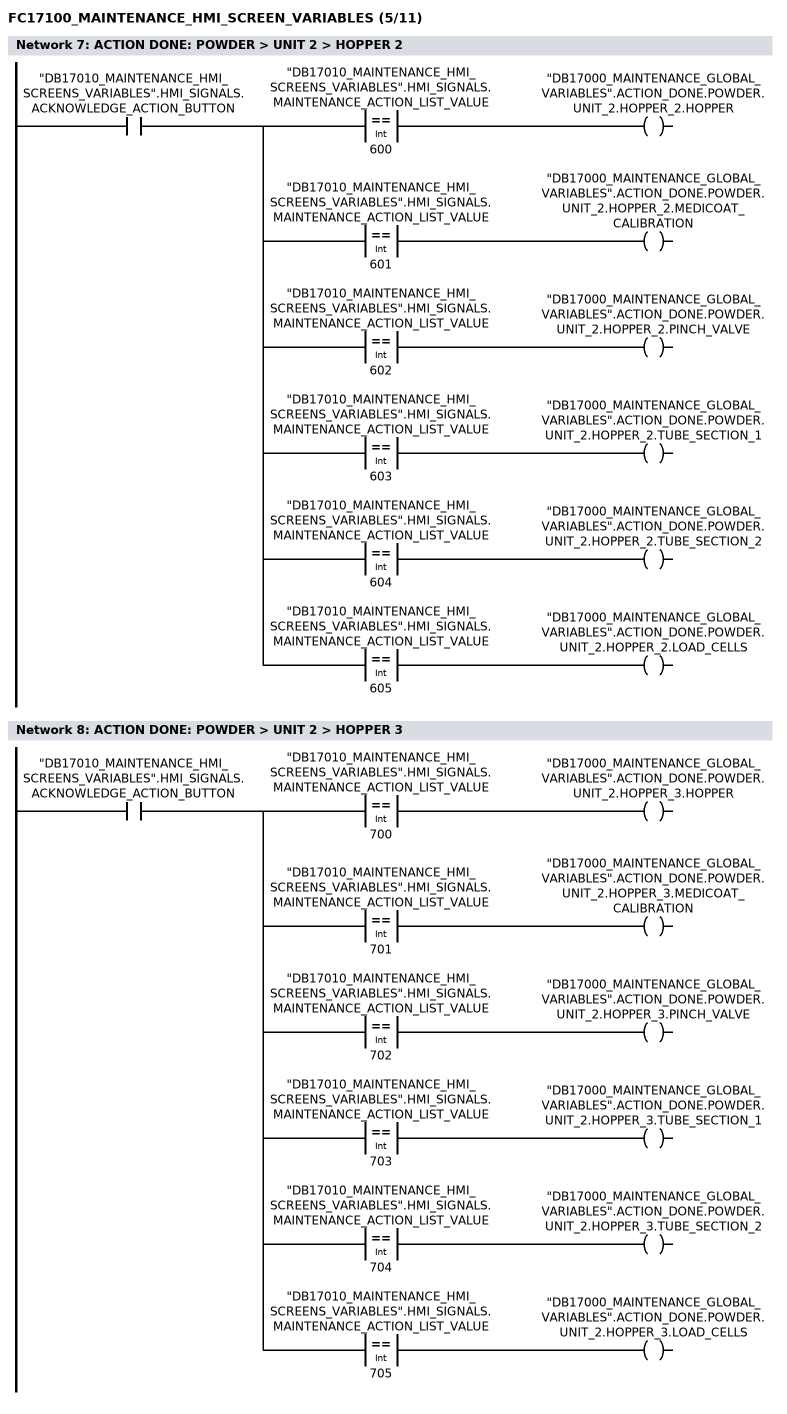
   RUNG wire#powerrail
      Contact( "DB17010_MAINTENANCE_HMI_SCREENS_VARIABLES".HMI_SIGNALS.ACKNOWLEDGE_ACTION_BUTTON )
      wire#w1
      { S7_Templates := "SrcType := Int" } EQ_Contact(in1 := "DB17010_MAINTENANCE_HMI_SCREENS_VARIABLES".HMI_SIGNALS.MAINTENANCE_ACTION_LIST_VALUE, in2 := 600)
      Coil( "DB17000_MAINTENANCE_GLOBAL_VARIABLES".ACTION_DONE.POWDER.UNIT_2.HOPPER_2.HOPPER )
   END_RUNG
   RUNG wire#w1
      { S7_Templates := "SrcType := Int" } EQ_Contact(in1 := "DB17010_MAINTENANCE_HMI_SCREENS_VARIABLES".HMI_SIGNALS.MAINTENANCE_ACTION_LIST_VALUE, in2 := 601)
      Coil( "DB17000_MAINTENANCE_GLOBAL_VARIABLES".ACTION_DONE.POWDER.UNIT_2.HOPPER_2.MEDICOAT_CALIBRATION )
   END_RUNG
   RUNG wire#w1
      { S7_Templates := "SrcType := Int" } EQ_Contact(in1 := "DB17010_MAINTENANCE_HMI_SCREENS_VARIABLES".HMI_SIGNALS.MAINTENANCE_ACTION_LIST_VALUE, in2 := 602)
      Coil( "DB17000_MAINTENANCE_GLOBAL_VARIABLES".ACTION_DONE.POWDER.UNIT_2.HOPPER_2.PINCH_VALVE )
   END_RUNG
   RUNG wire#w1
      { S7_Templates := "SrcType := Int" } EQ_Contact(in1 := "DB17010_MAINTENANCE_HMI_SCREENS_VARIABLES".HMI_SIGNALS.MAINTENANCE_ACTION_LIST_VALUE, in2 := 603)
      Coil( "DB17000_MAINTENANCE_GLOBAL_VARIABLES".ACTION_DONE.POWDER.UNIT_2.HOPPER_2.TUBE_SECTION_1 )
   END_RUNG
   RUNG wire#w1
      { S7_Templates := "SrcType := Int" } EQ_Contact(in1 := "DB17010_MAINTENANCE_HMI_SCREENS_VARIABLES".HMI_SIGNALS.MAINTENANCE_ACTION_LIST_VALUE, in2 := 604)
      Coil( "DB17000_MAINTENANCE_GLOBAL_VARIABLES".ACTION_DONE.POWDER.UNIT_2.HOPPER_2.TUBE_SECTION_2 )
   END_RUNG
   RUNG wire#w1
      { S7_Templates := "SrcType := Int" } EQ_Contact(in1 := "DB17010_MAINTENANCE_HMI_SCREENS_VARIABLES".HMI_SIGNALS.MAINTENANCE_ACTION_LIST_VALUE, in2 := 605)
      Coil( "DB17000_MAINTENANCE_GLOBAL_VARIABLES".ACTION_DONE.POWDER.UNIT_2.HOPPER_2.LOAD_CELLS )
   END_RUNG
   // the same network as SCL:
   "DB17000_MAINTENANCE_GLOBAL_VARIABLES".ACTION_DONE.POWDER.UNIT_2.HOPPER_2.HOPPER := "DB17010_MAINTENANCE_HMI_SCREENS_VARIABLES".HMI_SIGNALS.ACKNOWLEDGE_ACTION_BUTTON AND ("DB17010_MAINTENANCE_HMI_SCREENS_VARIABLES".HMI_SIGNALS.MAINTENANCE_ACTION_LIST_VALUE = 600);
   "DB17000_MAINTENANCE_GLOBAL_VARIABLES".ACTION_DONE.POWDER.UNIT_2.HOPPER_2.MEDICOAT_CALIBRATION := "DB17010_MAINTENANCE_HMI_SCREENS_VARIABLES".HMI_SIGNALS.ACKNOWLEDGE_ACTION_BUTTON AND ("DB17010_MAINTENANCE_HMI_SCREENS_VARIABLES".HMI_SIGNALS.MAINTENANCE_ACTION_LIST_VALUE = 601);
   "DB17000_MAINTENANCE_GLOBAL_VARIABLES".ACTION_DONE.POWDER.UNIT_2.HOPPER_2.PINCH_VALVE := "DB17010_MAINTENANCE_HMI_SCREENS_VARIABLES".HMI_SIGNALS.ACKNOWLEDGE_ACTION_BUTTON AND ("DB17010_MAINTENANCE_HMI_SCREENS_VARIABLES".HMI_SIGNALS.MAINTENANCE_ACTION_LIST_VALUE = 602);
   "DB17000_MAINTENANCE_GLOBAL_VARIABLES".ACTION_DONE.POWDER.UNIT_2.HOPPER_2.TUBE_SECTION_1 := "DB17010_MAINTENANCE_HMI_SCREENS_VARIABLES".HMI_SIGNALS.ACKNOWLEDGE_ACTION_BUTTON AND ("DB17010_MAINTENANCE_HMI_SCREENS_VARIABLES".HMI_SIGNALS.MAINTENANCE_ACTION_LIST_VALUE = 603);
   "DB17000_MAINTENANCE_GLOBAL_VARIABLES".ACTION_DONE.POWDER.UNIT_2.HOPPER_2.TUBE_SECTION_2 := "DB17010_MAINTENANCE_HMI_SCREENS_VARIABLES".HMI_SIGNALS.ACKNOWLEDGE_ACTION_BUTTON AND ("DB17010_MAINTENANCE_HMI_SCREENS_VARIABLES".HMI_SIGNALS.MAINTENANCE_ACTION_LIST_VALUE = 604);
   "DB17000_MAINTENANCE_GLOBAL_VARIABLES".ACTION_DONE.POWDER.UNIT_2.HOPPER_2.LOAD_CELLS := "DB17010_MAINTENANCE_HMI_SCREENS_VARIABLES".HMI_SIGNALS.ACKNOWLEDGE_ACTION_BUTTON AND ("DB17010_MAINTENANCE_HMI_SCREENS_VARIABLES".HMI_SIGNALS.MAINTENANCE_ACTION_LIST_VALUE = 605);
END_REGION

REGION Network 8: ACTION DONE: POWDER > UNIT 2 > HOPPER 3
   RUNG wire#powerrail
      Contact( "DB17010_MAINTENANCE_HMI_SCREENS_VARIABLES".HMI_SIGNALS.ACKNOWLEDGE_ACTION_BUTTON )
      wire#w1
      { S7_Templates := "SrcType := Int" } EQ_Contact(in1 := "DB17010_MAINTENANCE_HMI_SCREENS_VARIABLES".HMI_SIGNALS.MAINTENANCE_ACTION_LIST_VALUE, in2 := 700)
      Coil( "DB17000_MAINTENANCE_GLOBAL_VARIABLES".ACTION_DONE.POWDER.UNIT_2.HOPPER_3.HOPPER )
   END_RUNG
   RUNG wire#w1
      { S7_Templates := "SrcType := Int" } EQ_Contact(in1 := "DB17010_MAINTENANCE_HMI_SCREENS_VARIABLES".HMI_SIGNALS.MAINTENANCE_ACTION_LIST_VALUE, in2 := 701)
      Coil( "DB17000_MAINTENANCE_GLOBAL_VARIABLES".ACTION_DONE.POWDER.UNIT_2.HOPPER_3.MEDICOAT_CALIBRATION )
   END_RUNG
   RUNG wire#w1
      { S7_Templates := "SrcType := Int" } EQ_Contact(in1 := "DB17010_MAINTENANCE_HMI_SCREENS_VARIABLES".HMI_SIGNALS.MAINTENANCE_ACTION_LIST_VALUE, in2 := 702)
      Coil( "DB17000_MAINTENANCE_GLOBAL_VARIABLES".ACTION_DONE.POWDER.UNIT_2.HOPPER_3.PINCH_VALVE )
   END_RUNG
   RUNG wire#w1
      { S7_Templates := "SrcType := Int" } EQ_Contact(in1 := "DB17010_MAINTENANCE_HMI_SCREENS_VARIABLES".HMI_SIGNALS.MAINTENANCE_ACTION_LIST_VALUE, in2 := 703)
      Coil( "DB17000_MAINTENANCE_GLOBAL_VARIABLES".ACTION_DONE.POWDER.UNIT_2.HOPPER_3.TUBE_SECTION_1 )
   END_RUNG
   RUNG wire#w1
      { S7_Templates := "SrcType := Int" } EQ_Contact(in1 := "DB17010_MAINTENANCE_HMI_SCREENS_VARIABLES".HMI_SIGNALS.MAINTENANCE_ACTION_LIST_VALUE, in2 := 704)
      Coil( "DB17000_MAINTENANCE_GLOBAL_VARIABLES".ACTION_DONE.POWDER.UNIT_2.HOPPER_3.TUBE_SECTION_2 )
   END_RUNG
   RUNG wire#w1
      { S7_Templates := "SrcType := Int" } EQ_Contact(in1 := "DB17010_MAINTENANCE_HMI_SCREENS_VARIABLES".HMI_SIGNALS.MAINTENANCE_ACTION_LIST_VALUE, in2 := 705)
      Coil( "DB17000_MAINTENANCE_GLOBAL_VARIABLES".ACTION_DONE.POWDER.UNIT_2.HOPPER_3.LOAD_CELLS )
   END_RUNG
   // the same network as SCL:
   "DB17000_MAINTENANCE_GLOBAL_VARIABLES".ACTION_DONE.POWDER.UNIT_2.HOPPER_3.HOPPER := "DB17010_MAINTENANCE_HMI_SCREENS_VARIABLES".HMI_SIGNALS.ACKNOWLEDGE_ACTION_BUTTON AND ("DB17010_MAINTENANCE_HMI_SCREENS_VARIABLES".HMI_SIGNALS.MAINTENANCE_ACTION_LIST_VALUE = 700);
   "DB17000_MAINTENANCE_GLOBAL_VARIABLES".ACTION_DONE.POWDER.UNIT_2.HOPPER_3.MEDICOAT_CALIBRATION := "DB17010_MAINTENANCE_HMI_SCREENS_VARIABLES".HMI_SIGNALS.ACKNOWLEDGE_ACTION_BUTTON AND ("DB17010_MAINTENANCE_HMI_SCREENS_VARIABLES".HMI_SIGNALS.MAINTENANCE_ACTION_LIST_VALUE = 701);
   "DB17000_MAINTENANCE_GLOBAL_VARIABLES".ACTION_DONE.POWDER.UNIT_2.HOPPER_3.PINCH_VALVE := "DB17010_MAINTENANCE_HMI_SCREENS_VARIABLES".HMI_SIGNALS.ACKNOWLEDGE_ACTION_BUTTON AND ("DB17010_MAINTENANCE_HMI_SCREENS_VARIABLES".HMI_SIGNALS.MAINTENANCE_ACTION_LIST_VALUE = 702);
   "DB17000_MAINTENANCE_GLOBAL_VARIABLES".ACTION_DONE.POWDER.UNIT_2.HOPPER_3.TUBE_SECTION_1 := "DB17010_MAINTENANCE_HMI_SCREENS_VARIABLES".HMI_SIGNALS.ACKNOWLEDGE_ACTION_BUTTON AND ("DB17010_MAINTENANCE_HMI_SCREENS_VARIABLES".HMI_SIGNALS.MAINTENANCE_ACTION_LIST_VALUE = 703);
   "DB17000_MAINTENANCE_GLOBAL_VARIABLES".ACTION_DONE.POWDER.UNIT_2.HOPPER_3.TUBE_SECTION_2 := "DB17010_MAINTENANCE_HMI_SCREENS_VARIABLES".HMI_SIGNALS.ACKNOWLEDGE_ACTION_BUTTON AND ("DB17010_MAINTENANCE_HMI_SCREENS_VARIABLES".HMI_SIGNALS.MAINTENANCE_ACTION_LIST_VALUE = 704);
   "DB17000_MAINTENANCE_GLOBAL_VARIABLES".ACTION_DONE.POWDER.UNIT_2.HOPPER_3.LOAD_CELLS := "DB17010_MAINTENANCE_HMI_SCREENS_VARIABLES".HMI_SIGNALS.ACKNOWLEDGE_ACTION_BUTTON AND ("DB17010_MAINTENANCE_HMI_SCREENS_VARIABLES".HMI_SIGNALS.MAINTENANCE_ACTION_LIST_VALUE = 705);
END_REGION

REGION Network 9: ACTION DONE: POWDER > UNIT 2 > FEEDER 1
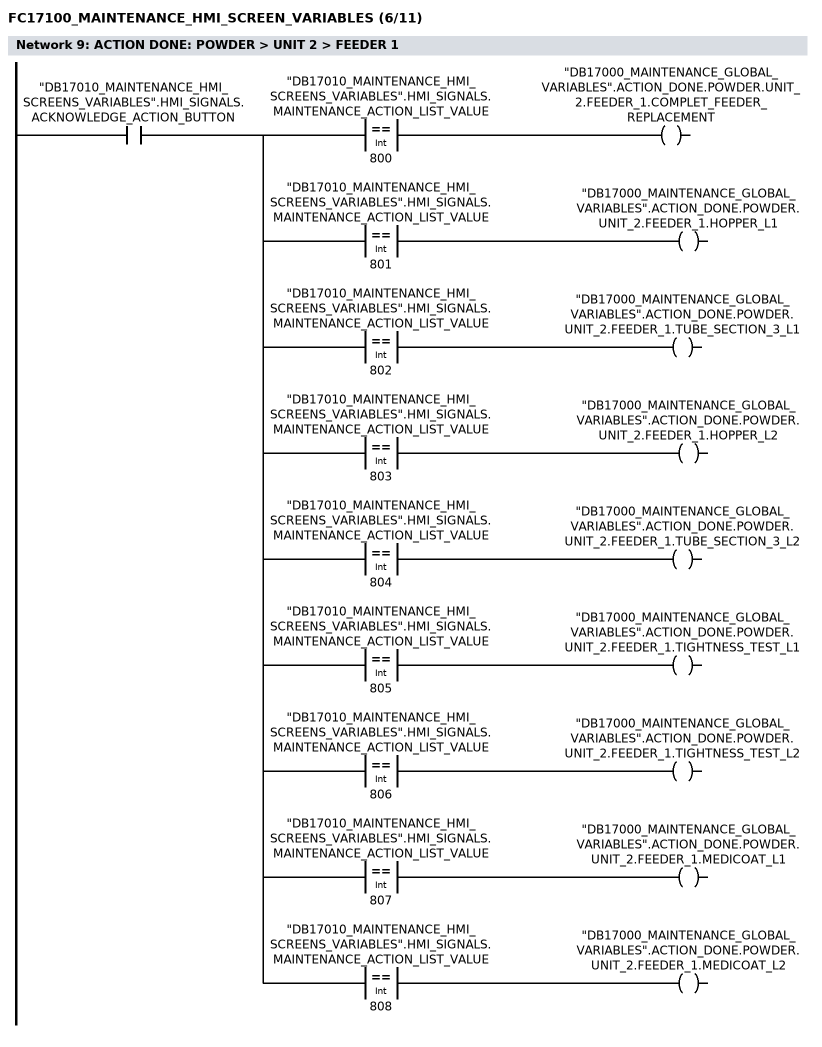
   RUNG wire#powerrail
      Contact( "DB17010_MAINTENANCE_HMI_SCREENS_VARIABLES".HMI_SIGNALS.ACKNOWLEDGE_ACTION_BUTTON )
      wire#w1
      { S7_Templates := "SrcType := Int" } EQ_Contact(in1 := "DB17010_MAINTENANCE_HMI_SCREENS_VARIABLES".HMI_SIGNALS.MAINTENANCE_ACTION_LIST_VALUE, in2 := 800)
      Coil( "DB17000_MAINTENANCE_GLOBAL_VARIABLES".ACTION_DONE.POWDER.UNIT_2.FEEDER_1.COMPLET_FEEDER_REPLACEMENT )
   END_RUNG
   RUNG wire#w1
      { S7_Templates := "SrcType := Int" } EQ_Contact(in1 := "DB17010_MAINTENANCE_HMI_SCREENS_VARIABLES".HMI_SIGNALS.MAINTENANCE_ACTION_LIST_VALUE, in2 := 801)
      Coil( "DB17000_MAINTENANCE_GLOBAL_VARIABLES".ACTION_DONE.POWDER.UNIT_2.FEEDER_1.HOPPER_L1 )
   END_RUNG
   RUNG wire#w1
      { S7_Templates := "SrcType := Int" } EQ_Contact(in1 := "DB17010_MAINTENANCE_HMI_SCREENS_VARIABLES".HMI_SIGNALS.MAINTENANCE_ACTION_LIST_VALUE, in2 := 802)
      Coil( "DB17000_MAINTENANCE_GLOBAL_VARIABLES".ACTION_DONE.POWDER.UNIT_2.FEEDER_1.TUBE_SECTION_3_L1 )
   END_RUNG
   RUNG wire#w1
      { S7_Templates := "SrcType := Int" } EQ_Contact(in1 := "DB17010_MAINTENANCE_HMI_SCREENS_VARIABLES".HMI_SIGNALS.MAINTENANCE_ACTION_LIST_VALUE, in2 := 803)
      Coil( "DB17000_MAINTENANCE_GLOBAL_VARIABLES".ACTION_DONE.POWDER.UNIT_2.FEEDER_1.HOPPER_L2 )
   END_RUNG
   RUNG wire#w1
      { S7_Templates := "SrcType := Int" } EQ_Contact(in1 := "DB17010_MAINTENANCE_HMI_SCREENS_VARIABLES".HMI_SIGNALS.MAINTENANCE_ACTION_LIST_VALUE, in2 := 804)
      Coil( "DB17000_MAINTENANCE_GLOBAL_VARIABLES".ACTION_DONE.POWDER.UNIT_2.FEEDER_1.TUBE_SECTION_3_L2 )
   END_RUNG
   RUNG wire#w1
      { S7_Templates := "SrcType := Int" } EQ_Contact(in1 := "DB17010_MAINTENANCE_HMI_SCREENS_VARIABLES".HMI_SIGNALS.MAINTENANCE_ACTION_LIST_VALUE, in2 := 805)
      Coil( "DB17000_MAINTENANCE_GLOBAL_VARIABLES".ACTION_DONE.POWDER.UNIT_2.FEEDER_1.TIGHTNESS_TEST_L1 )
   END_RUNG
   RUNG wire#w1
      { S7_Templates := "SrcType := Int" } EQ_Contact(in1 := "DB17010_MAINTENANCE_HMI_SCREENS_VARIABLES".HMI_SIGNALS.MAINTENANCE_ACTION_LIST_VALUE, in2 := 806)
      Coil( "DB17000_MAINTENANCE_GLOBAL_VARIABLES".ACTION_DONE.POWDER.UNIT_2.FEEDER_1.TIGHTNESS_TEST_L2 )
   END_RUNG
   RUNG wire#w1
      { S7_Templates := "SrcType := Int" } EQ_Contact(in1 := "DB17010_MAINTENANCE_HMI_SCREENS_VARIABLES".HMI_SIGNALS.MAINTENANCE_ACTION_LIST_VALUE, in2 := 807)
      Coil( "DB17000_MAINTENANCE_GLOBAL_VARIABLES".ACTION_DONE.POWDER.UNIT_2.FEEDER_1.MEDICOAT_L1 )
   END_RUNG
   RUNG wire#w1
      { S7_Templates := "SrcType := Int" } EQ_Contact(in1 := "DB17010_MAINTENANCE_HMI_SCREENS_VARIABLES".HMI_SIGNALS.MAINTENANCE_ACTION_LIST_VALUE, in2 := 808)
      Coil( "DB17000_MAINTENANCE_GLOBAL_VARIABLES".ACTION_DONE.POWDER.UNIT_2.FEEDER_1.MEDICOAT_L2 )
   END_RUNG
   // the same network as SCL:
   "DB17000_MAINTENANCE_GLOBAL_VARIABLES".ACTION_DONE.POWDER.UNIT_2.FEEDER_1.COMPLET_FEEDER_REPLACEMENT := "DB17010_MAINTENANCE_HMI_SCREENS_VARIABLES".HMI_SIGNALS.ACKNOWLEDGE_ACTION_BUTTON AND ("DB17010_MAINTENANCE_HMI_SCREENS_VARIABLES".HMI_SIGNALS.MAINTENANCE_ACTION_LIST_VALUE = 800);
   "DB17000_MAINTENANCE_GLOBAL_VARIABLES".ACTION_DONE.POWDER.UNIT_2.FEEDER_1.HOPPER_L1 := "DB17010_MAINTENANCE_HMI_SCREENS_VARIABLES".HMI_SIGNALS.ACKNOWLEDGE_ACTION_BUTTON AND ("DB17010_MAINTENANCE_HMI_SCREENS_VARIABLES".HMI_SIGNALS.MAINTENANCE_ACTION_LIST_VALUE = 801);
   "DB17000_MAINTENANCE_GLOBAL_VARIABLES".ACTION_DONE.POWDER.UNIT_2.FEEDER_1.TUBE_SECTION_3_L1 := "DB17010_MAINTENANCE_HMI_SCREENS_VARIABLES".HMI_SIGNALS.ACKNOWLEDGE_ACTION_BUTTON AND ("DB17010_MAINTENANCE_HMI_SCREENS_VARIABLES".HMI_SIGNALS.MAINTENANCE_ACTION_LIST_VALUE = 802);
   "DB17000_MAINTENANCE_GLOBAL_VARIABLES".ACTION_DONE.POWDER.UNIT_2.FEEDER_1.HOPPER_L2 := "DB17010_MAINTENANCE_HMI_SCREENS_VARIABLES".HMI_SIGNALS.ACKNOWLEDGE_ACTION_BUTTON AND ("DB17010_MAINTENANCE_HMI_SCREENS_VARIABLES".HMI_SIGNALS.MAINTENANCE_ACTION_LIST_VALUE = 803);
   "DB17000_MAINTENANCE_GLOBAL_VARIABLES".ACTION_DONE.POWDER.UNIT_2.FEEDER_1.TUBE_SECTION_3_L2 := "DB17010_MAINTENANCE_HMI_SCREENS_VARIABLES".HMI_SIGNALS.ACKNOWLEDGE_ACTION_BUTTON AND ("DB17010_MAINTENANCE_HMI_SCREENS_VARIABLES".HMI_SIGNALS.MAINTENANCE_ACTION_LIST_VALUE = 804);
   "DB17000_MAINTENANCE_GLOBAL_VARIABLES".ACTION_DONE.POWDER.UNIT_2.FEEDER_1.TIGHTNESS_TEST_L1 := "DB17010_MAINTENANCE_HMI_SCREENS_VARIABLES".HMI_SIGNALS.ACKNOWLEDGE_ACTION_BUTTON AND ("DB17010_MAINTENANCE_HMI_SCREENS_VARIABLES".HMI_SIGNALS.MAINTENANCE_ACTION_LIST_VALUE = 805);
   "DB17000_MAINTENANCE_GLOBAL_VARIABLES".ACTION_DONE.POWDER.UNIT_2.FEEDER_1.TIGHTNESS_TEST_L2 := "DB17010_MAINTENANCE_HMI_SCREENS_VARIABLES".HMI_SIGNALS.ACKNOWLEDGE_ACTION_BUTTON AND ("DB17010_MAINTENANCE_HMI_SCREENS_VARIABLES".HMI_SIGNALS.MAINTENANCE_ACTION_LIST_VALUE = 806);
   "DB17000_MAINTENANCE_GLOBAL_VARIABLES".ACTION_DONE.POWDER.UNIT_2.FEEDER_1.MEDICOAT_L1 := "DB17010_MAINTENANCE_HMI_SCREENS_VARIABLES".HMI_SIGNALS.ACKNOWLEDGE_ACTION_BUTTON AND ("DB17010_MAINTENANCE_HMI_SCREENS_VARIABLES".HMI_SIGNALS.MAINTENANCE_ACTION_LIST_VALUE = 807);
   "DB17000_MAINTENANCE_GLOBAL_VARIABLES".ACTION_DONE.POWDER.UNIT_2.FEEDER_1.MEDICOAT_L2 := "DB17010_MAINTENANCE_HMI_SCREENS_VARIABLES".HMI_SIGNALS.ACKNOWLEDGE_ACTION_BUTTON AND ("DB17010_MAINTENANCE_HMI_SCREENS_VARIABLES".HMI_SIGNALS.MAINTENANCE_ACTION_LIST_VALUE = 808);
END_REGION

REGION Network 10: ACTION DONE: POWDER > UNIT 2 > FEEDER 2
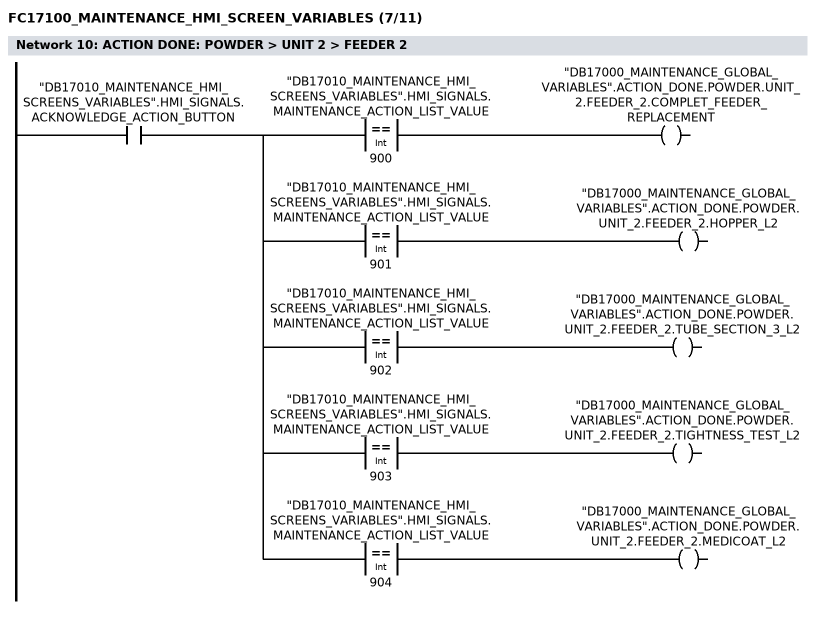
   RUNG wire#powerrail
      Contact( "DB17010_MAINTENANCE_HMI_SCREENS_VARIABLES".HMI_SIGNALS.ACKNOWLEDGE_ACTION_BUTTON )
      wire#w1
      { S7_Templates := "SrcType := Int" } EQ_Contact(in1 := "DB17010_MAINTENANCE_HMI_SCREENS_VARIABLES".HMI_SIGNALS.MAINTENANCE_ACTION_LIST_VALUE, in2 := 900)
      Coil( "DB17000_MAINTENANCE_GLOBAL_VARIABLES".ACTION_DONE.POWDER.UNIT_2.FEEDER_2.COMPLET_FEEDER_REPLACEMENT )
   END_RUNG
   RUNG wire#w1
      { S7_Templates := "SrcType := Int" } EQ_Contact(in1 := "DB17010_MAINTENANCE_HMI_SCREENS_VARIABLES".HMI_SIGNALS.MAINTENANCE_ACTION_LIST_VALUE, in2 := 901)
      Coil( "DB17000_MAINTENANCE_GLOBAL_VARIABLES".ACTION_DONE.POWDER.UNIT_2.FEEDER_2.HOPPER_L2 )
   END_RUNG
   RUNG wire#w1
      { S7_Templates := "SrcType := Int" } EQ_Contact(in1 := "DB17010_MAINTENANCE_HMI_SCREENS_VARIABLES".HMI_SIGNALS.MAINTENANCE_ACTION_LIST_VALUE, in2 := 902)
      Coil( "DB17000_MAINTENANCE_GLOBAL_VARIABLES".ACTION_DONE.POWDER.UNIT_2.FEEDER_2.TUBE_SECTION_3_L2 )
   END_RUNG
   RUNG wire#w1
      { S7_Templates := "SrcType := Int" } EQ_Contact(in1 := "DB17010_MAINTENANCE_HMI_SCREENS_VARIABLES".HMI_SIGNALS.MAINTENANCE_ACTION_LIST_VALUE, in2 := 903)
      Coil( "DB17000_MAINTENANCE_GLOBAL_VARIABLES".ACTION_DONE.POWDER.UNIT_2.FEEDER_2.TIGHTNESS_TEST_L2 )
   END_RUNG
   RUNG wire#w1
      { S7_Templates := "SrcType := Int" } EQ_Contact(in1 := "DB17010_MAINTENANCE_HMI_SCREENS_VARIABLES".HMI_SIGNALS.MAINTENANCE_ACTION_LIST_VALUE, in2 := 904)
      Coil( "DB17000_MAINTENANCE_GLOBAL_VARIABLES".ACTION_DONE.POWDER.UNIT_2.FEEDER_2.MEDICOAT_L2 )
   END_RUNG
   // the same network as SCL:
   "DB17000_MAINTENANCE_GLOBAL_VARIABLES".ACTION_DONE.POWDER.UNIT_2.FEEDER_2.COMPLET_FEEDER_REPLACEMENT := "DB17010_MAINTENANCE_HMI_SCREENS_VARIABLES".HMI_SIGNALS.ACKNOWLEDGE_ACTION_BUTTON AND ("DB17010_MAINTENANCE_HMI_SCREENS_VARIABLES".HMI_SIGNALS.MAINTENANCE_ACTION_LIST_VALUE = 900);
   "DB17000_MAINTENANCE_GLOBAL_VARIABLES".ACTION_DONE.POWDER.UNIT_2.FEEDER_2.HOPPER_L2 := "DB17010_MAINTENANCE_HMI_SCREENS_VARIABLES".HMI_SIGNALS.ACKNOWLEDGE_ACTION_BUTTON AND ("DB17010_MAINTENANCE_HMI_SCREENS_VARIABLES".HMI_SIGNALS.MAINTENANCE_ACTION_LIST_VALUE = 901);
   "DB17000_MAINTENANCE_GLOBAL_VARIABLES".ACTION_DONE.POWDER.UNIT_2.FEEDER_2.TUBE_SECTION_3_L2 := "DB17010_MAINTENANCE_HMI_SCREENS_VARIABLES".HMI_SIGNALS.ACKNOWLEDGE_ACTION_BUTTON AND ("DB17010_MAINTENANCE_HMI_SCREENS_VARIABLES".HMI_SIGNALS.MAINTENANCE_ACTION_LIST_VALUE = 902);
   "DB17000_MAINTENANCE_GLOBAL_VARIABLES".ACTION_DONE.POWDER.UNIT_2.FEEDER_2.TIGHTNESS_TEST_L2 := "DB17010_MAINTENANCE_HMI_SCREENS_VARIABLES".HMI_SIGNALS.ACKNOWLEDGE_ACTION_BUTTON AND ("DB17010_MAINTENANCE_HMI_SCREENS_VARIABLES".HMI_SIGNALS.MAINTENANCE_ACTION_LIST_VALUE = 903);
   "DB17000_MAINTENANCE_GLOBAL_VARIABLES".ACTION_DONE.POWDER.UNIT_2.FEEDER_2.MEDICOAT_L2 := "DB17010_MAINTENANCE_HMI_SCREENS_VARIABLES".HMI_SIGNALS.ACKNOWLEDGE_ACTION_BUTTON AND ("DB17010_MAINTENANCE_HMI_SCREENS_VARIABLES".HMI_SIGNALS.MAINTENANCE_ACTION_LIST_VALUE = 904);
END_REGION

REGION Network 11: ACTION DONE: MACHINE > UNIT 1 > GENERAL
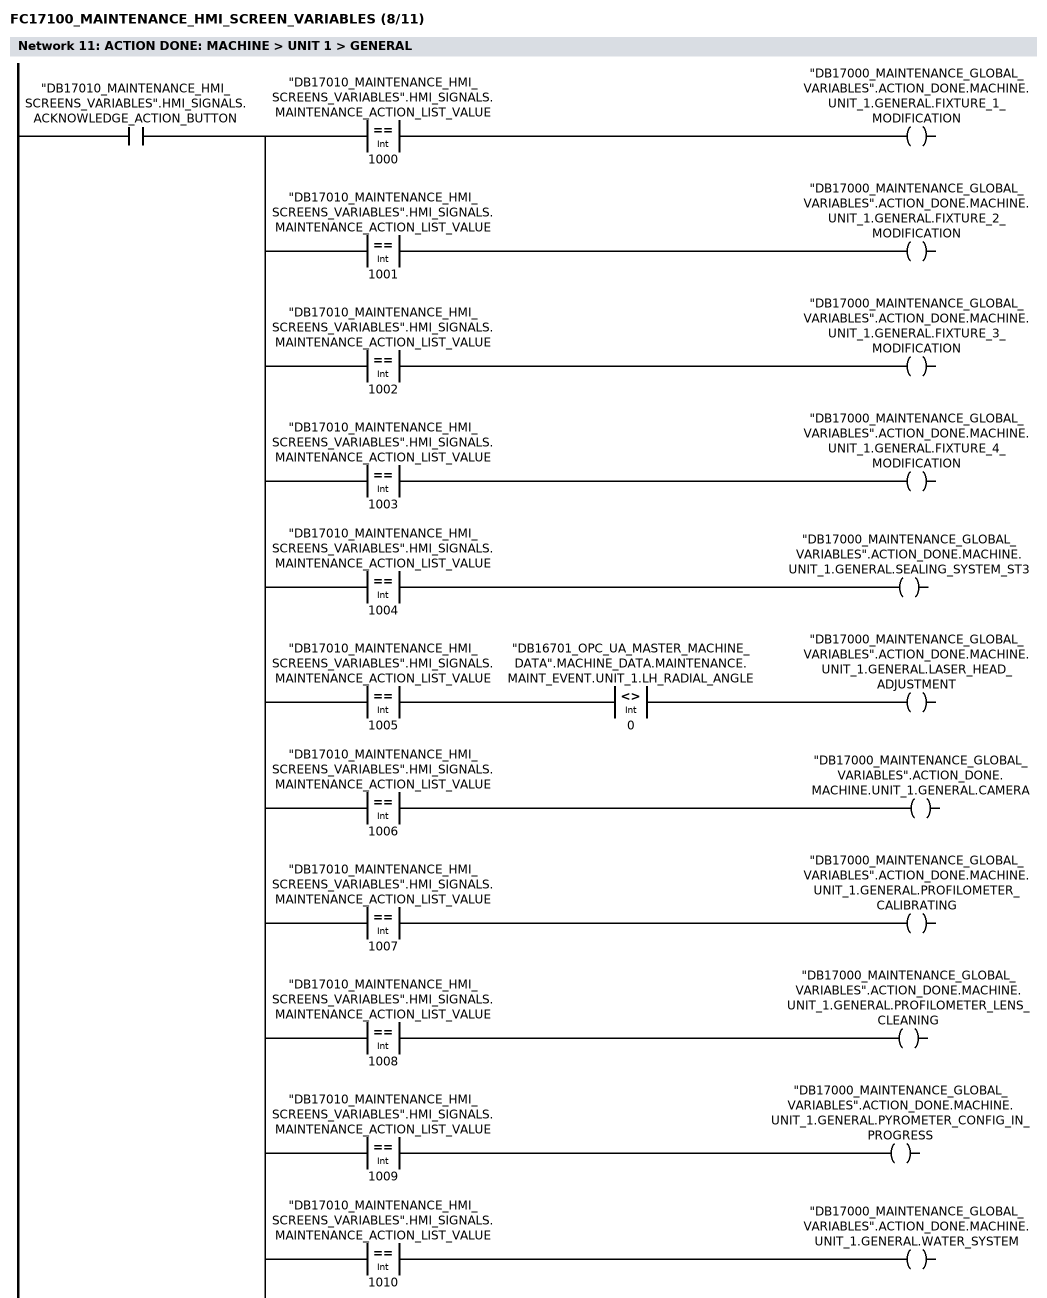
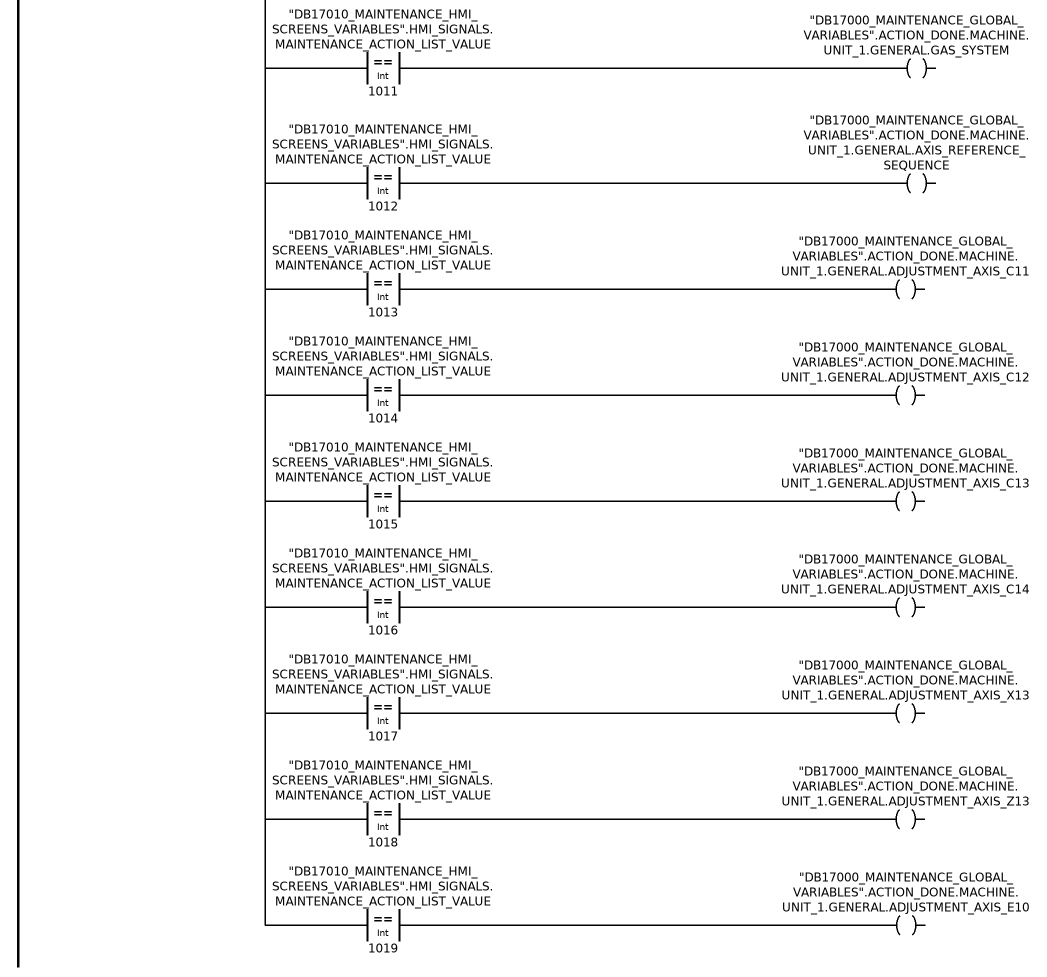
   RUNG wire#powerrail
      Contact( "DB17010_MAINTENANCE_HMI_SCREENS_VARIABLES".HMI_SIGNALS.ACKNOWLEDGE_ACTION_BUTTON )
      wire#w1
      { S7_Templates := "SrcType := Int" } EQ_Contact(in1 := "DB17010_MAINTENANCE_HMI_SCREENS_VARIABLES".HMI_SIGNALS.MAINTENANCE_ACTION_LIST_VALUE, in2 := 1000)
      Coil( "DB17000_MAINTENANCE_GLOBAL_VARIABLES".ACTION_DONE.MACHINE.UNIT_1.GENERAL.FIXTURE_1_MODIFICATION )
   END_RUNG
   RUNG wire#w1
      { S7_Templates := "SrcType := Int" } EQ_Contact(in1 := "DB17010_MAINTENANCE_HMI_SCREENS_VARIABLES".HMI_SIGNALS.MAINTENANCE_ACTION_LIST_VALUE, in2 := 1001)
      Coil( "DB17000_MAINTENANCE_GLOBAL_VARIABLES".ACTION_DONE.MACHINE.UNIT_1.GENERAL.FIXTURE_2_MODIFICATION )
   END_RUNG
   RUNG wire#w1
      { S7_Templates := "SrcType := Int" } EQ_Contact(in1 := "DB17010_MAINTENANCE_HMI_SCREENS_VARIABLES".HMI_SIGNALS.MAINTENANCE_ACTION_LIST_VALUE, in2 := 1002)
      Coil( "DB17000_MAINTENANCE_GLOBAL_VARIABLES".ACTION_DONE.MACHINE.UNIT_1.GENERAL.FIXTURE_3_MODIFICATION )
   END_RUNG
   RUNG wire#w1
      { S7_Templates := "SrcType := Int" } EQ_Contact(in1 := "DB17010_MAINTENANCE_HMI_SCREENS_VARIABLES".HMI_SIGNALS.MAINTENANCE_ACTION_LIST_VALUE, in2 := 1003)
      Coil( "DB17000_MAINTENANCE_GLOBAL_VARIABLES".ACTION_DONE.MACHINE.UNIT_1.GENERAL.FIXTURE_4_MODIFICATION )
   END_RUNG
   RUNG wire#w1
      { S7_Templates := "SrcType := Int" } EQ_Contact(in1 := "DB17010_MAINTENANCE_HMI_SCREENS_VARIABLES".HMI_SIGNALS.MAINTENANCE_ACTION_LIST_VALUE, in2 := 1004)
      Coil( "DB17000_MAINTENANCE_GLOBAL_VARIABLES".ACTION_DONE.MACHINE.UNIT_1.GENERAL.SEALING_SYSTEM_ST3 )
   END_RUNG
   RUNG wire#w1
      { S7_Templates := "SrcType := Int" } EQ_Contact(in1 := "DB17010_MAINTENANCE_HMI_SCREENS_VARIABLES".HMI_SIGNALS.MAINTENANCE_ACTION_LIST_VALUE, in2 := 1005)
      { S7_Templates := "SrcType := Int" } NE_Contact(in1 := "DB16701_OPC_UA_MASTER_MACHINE_DATA".MACHINE_DATA.MAINTENANCE.MAINT_EVENT.UNIT_1.LH_RADIAL_ANGLE, in2 := 0)
      Coil( "DB17000_MAINTENANCE_GLOBAL_VARIABLES".ACTION_DONE.MACHINE.UNIT_1.GENERAL.LASER_HEAD_ADJUSTMENT )
   END_RUNG
   RUNG wire#w1
      { S7_Templates := "SrcType := Int" } EQ_Contact(in1 := "DB17010_MAINTENANCE_HMI_SCREENS_VARIABLES".HMI_SIGNALS.MAINTENANCE_ACTION_LIST_VALUE, in2 := 1006)
      Coil( "DB17000_MAINTENANCE_GLOBAL_VARIABLES".ACTION_DONE.MACHINE.UNIT_1.GENERAL.CAMERA )
   END_RUNG
   RUNG wire#w1
      { S7_Templates := "SrcType := Int" } EQ_Contact(in1 := "DB17010_MAINTENANCE_HMI_SCREENS_VARIABLES".HMI_SIGNALS.MAINTENANCE_ACTION_LIST_VALUE, in2 := 1007)
      Coil( "DB17000_MAINTENANCE_GLOBAL_VARIABLES".ACTION_DONE.MACHINE.UNIT_1.GENERAL.PROFILOMETER_CALIBRATING )
   END_RUNG
   RUNG wire#w1
      { S7_Templates := "SrcType := Int" } EQ_Contact(in1 := "DB17010_MAINTENANCE_HMI_SCREENS_VARIABLES".HMI_SIGNALS.MAINTENANCE_ACTION_LIST_VALUE, in2 := 1008)
      Coil( "DB17000_MAINTENANCE_GLOBAL_VARIABLES".ACTION_DONE.MACHINE.UNIT_1.GENERAL.PROFILOMETER_LENS_CLEANING )
   END_RUNG
   RUNG wire#w1
      { S7_Templates := "SrcType := Int" } EQ_Contact(in1 := "DB17010_MAINTENANCE_HMI_SCREENS_VARIABLES".HMI_SIGNALS.MAINTENANCE_ACTION_LIST_VALUE, in2 := 1009)
      Coil( "DB17000_MAINTENANCE_GLOBAL_VARIABLES".ACTION_DONE.MACHINE.UNIT_1.GENERAL.PYROMETER_CONFIG_IN_PROGRESS )
   END_RUNG
   RUNG wire#w1
      { S7_Templates := "SrcType := Int" } EQ_Contact(in1 := "DB17010_MAINTENANCE_HMI_SCREENS_VARIABLES".HMI_SIGNALS.MAINTENANCE_ACTION_LIST_VALUE, in2 := 1010)
      Coil( "DB17000_MAINTENANCE_GLOBAL_VARIABLES".ACTION_DONE.MACHINE.UNIT_1.GENERAL.WATER_SYSTEM )
   END_RUNG
   RUNG wire#w1
      { S7_Templates := "SrcType := Int" } EQ_Contact(in1 := "DB17010_MAINTENANCE_HMI_SCREENS_VARIABLES".HMI_SIGNALS.MAINTENANCE_ACTION_LIST_VALUE, in2 := 1011)
      Coil( "DB17000_MAINTENANCE_GLOBAL_VARIABLES".ACTION_DONE.MACHINE.UNIT_1.GENERAL.GAS_SYSTEM )
   END_RUNG
   RUNG wire#w1
      { S7_Templates := "SrcType := Int" } EQ_Contact(in1 := "DB17010_MAINTENANCE_HMI_SCREENS_VARIABLES".HMI_SIGNALS.MAINTENANCE_ACTION_LIST_VALUE, in2 := 1012)
      Coil( "DB17000_MAINTENANCE_GLOBAL_VARIABLES".ACTION_DONE.MACHINE.UNIT_1.GENERAL.AXIS_REFERENCE_SEQUENCE )
   END_RUNG
   RUNG wire#w1
      { S7_Templates := "SrcType := Int" } EQ_Contact(in1 := "DB17010_MAINTENANCE_HMI_SCREENS_VARIABLES".HMI_SIGNALS.MAINTENANCE_ACTION_LIST_VALUE, in2 := 1013)
      Coil( "DB17000_MAINTENANCE_GLOBAL_VARIABLES".ACTION_DONE.MACHINE.UNIT_1.GENERAL.ADJUSTMENT_AXIS_C11 )
   END_RUNG
   RUNG wire#w1
      { S7_Templates := "SrcType := Int" } EQ_Contact(in1 := "DB17010_MAINTENANCE_HMI_SCREENS_VARIABLES".HMI_SIGNALS.MAINTENANCE_ACTION_LIST_VALUE, in2 := 1014)
      Coil( "DB17000_MAINTENANCE_GLOBAL_VARIABLES".ACTION_DONE.MACHINE.UNIT_1.GENERAL.ADJUSTMENT_AXIS_C12 )
   END_RUNG
   RUNG wire#w1
      { S7_Templates := "SrcType := Int" } EQ_Contact(in1 := "DB17010_MAINTENANCE_HMI_SCREENS_VARIABLES".HMI_SIGNALS.MAINTENANCE_ACTION_LIST_VALUE, in2 := 1015)
      Coil( "DB17000_MAINTENANCE_GLOBAL_VARIABLES".ACTION_DONE.MACHINE.UNIT_1.GENERAL.ADJUSTMENT_AXIS_C13 )
   END_RUNG
   RUNG wire#w1
      { S7_Templates := "SrcType := Int" } EQ_Contact(in1 := "DB17010_MAINTENANCE_HMI_SCREENS_VARIABLES".HMI_SIGNALS.MAINTENANCE_ACTION_LIST_VALUE, in2 := 1016)
      Coil( "DB17000_MAINTENANCE_GLOBAL_VARIABLES".ACTION_DONE.MACHINE.UNIT_1.GENERAL.ADJUSTMENT_AXIS_C14 )
   END_RUNG
   RUNG wire#w1
      { S7_Templates := "SrcType := Int" } EQ_Contact(in1 := "DB17010_MAINTENANCE_HMI_SCREENS_VARIABLES".HMI_SIGNALS.MAINTENANCE_ACTION_LIST_VALUE, in2 := 1017)
      Coil( "DB17000_MAINTENANCE_GLOBAL_VARIABLES".ACTION_DONE.MACHINE.UNIT_1.GENERAL.ADJUSTMENT_AXIS_X13 )
   END_RUNG
   RUNG wire#w1
      { S7_Templates := "SrcType := Int" } EQ_Contact(in1 := "DB17010_MAINTENANCE_HMI_SCREENS_VARIABLES".HMI_SIGNALS.MAINTENANCE_ACTION_LIST_VALUE, in2 := 1018)
      Coil( "DB17000_MAINTENANCE_GLOBAL_VARIABLES".ACTION_DONE.MACHINE.UNIT_1.GENERAL.ADJUSTMENT_AXIS_Z13 )
   END_RUNG
   RUNG wire#w1
      { S7_Templates := "SrcType := Int" } EQ_Contact(in1 := "DB17010_MAINTENANCE_HMI_SCREENS_VARIABLES".HMI_SIGNALS.MAINTENANCE_ACTION_LIST_VALUE, in2 := 1019)
      Coil( "DB17000_MAINTENANCE_GLOBAL_VARIABLES".ACTION_DONE.MACHINE.UNIT_1.GENERAL.ADJUSTMENT_AXIS_E10 )
   END_RUNG
   // the same network as SCL:
   "DB17000_MAINTENANCE_GLOBAL_VARIABLES".ACTION_DONE.MACHINE.UNIT_1.GENERAL.FIXTURE_1_MODIFICATION := "DB17010_MAINTENANCE_HMI_SCREENS_VARIABLES".HMI_SIGNALS.ACKNOWLEDGE_ACTION_BUTTON AND ("DB17010_MAINTENANCE_HMI_SCREENS_VARIABLES".HMI_SIGNALS.MAINTENANCE_ACTION_LIST_VALUE = 1000);
   "DB17000_MAINTENANCE_GLOBAL_VARIABLES".ACTION_DONE.MACHINE.UNIT_1.GENERAL.FIXTURE_2_MODIFICATION := "DB17010_MAINTENANCE_HMI_SCREENS_VARIABLES".HMI_SIGNALS.ACKNOWLEDGE_ACTION_BUTTON AND ("DB17010_MAINTENANCE_HMI_SCREENS_VARIABLES".HMI_SIGNALS.MAINTENANCE_ACTION_LIST_VALUE = 1001);
   "DB17000_MAINTENANCE_GLOBAL_VARIABLES".ACTION_DONE.MACHINE.UNIT_1.GENERAL.FIXTURE_3_MODIFICATION := "DB17010_MAINTENANCE_HMI_SCREENS_VARIABLES".HMI_SIGNALS.ACKNOWLEDGE_ACTION_BUTTON AND ("DB17010_MAINTENANCE_HMI_SCREENS_VARIABLES".HMI_SIGNALS.MAINTENANCE_ACTION_LIST_VALUE = 1002);
   "DB17000_MAINTENANCE_GLOBAL_VARIABLES".ACTION_DONE.MACHINE.UNIT_1.GENERAL.FIXTURE_4_MODIFICATION := "DB17010_MAINTENANCE_HMI_SCREENS_VARIABLES".HMI_SIGNALS.ACKNOWLEDGE_ACTION_BUTTON AND ("DB17010_MAINTENANCE_HMI_SCREENS_VARIABLES".HMI_SIGNALS.MAINTENANCE_ACTION_LIST_VALUE = 1003);
   "DB17000_MAINTENANCE_GLOBAL_VARIABLES".ACTION_DONE.MACHINE.UNIT_1.GENERAL.SEALING_SYSTEM_ST3 := "DB17010_MAINTENANCE_HMI_SCREENS_VARIABLES".HMI_SIGNALS.ACKNOWLEDGE_ACTION_BUTTON AND ("DB17010_MAINTENANCE_HMI_SCREENS_VARIABLES".HMI_SIGNALS.MAINTENANCE_ACTION_LIST_VALUE = 1004);
   "DB17000_MAINTENANCE_GLOBAL_VARIABLES".ACTION_DONE.MACHINE.UNIT_1.GENERAL.LASER_HEAD_ADJUSTMENT := "DB17010_MAINTENANCE_HMI_SCREENS_VARIABLES".HMI_SIGNALS.ACKNOWLEDGE_ACTION_BUTTON AND ("DB17010_MAINTENANCE_HMI_SCREENS_VARIABLES".HMI_SIGNALS.MAINTENANCE_ACTION_LIST_VALUE = 1005) AND ("DB16701_OPC_UA_MASTER_MACHINE_DATA".MACHINE_DATA.MAINTENANCE.MAINT_EVENT.UNIT_1.LH_RADIAL_ANGLE <> 0);
   "DB17000_MAINTENANCE_GLOBAL_VARIABLES".ACTION_DONE.MACHINE.UNIT_1.GENERAL.CAMERA := "DB17010_MAINTENANCE_HMI_SCREENS_VARIABLES".HMI_SIGNALS.ACKNOWLEDGE_ACTION_BUTTON AND ("DB17010_MAINTENANCE_HMI_SCREENS_VARIABLES".HMI_SIGNALS.MAINTENANCE_ACTION_LIST_VALUE = 1006);
   "DB17000_MAINTENANCE_GLOBAL_VARIABLES".ACTION_DONE.MACHINE.UNIT_1.GENERAL.PROFILOMETER_CALIBRATING := "DB17010_MAINTENANCE_HMI_SCREENS_VARIABLES".HMI_SIGNALS.ACKNOWLEDGE_ACTION_BUTTON AND ("DB17010_MAINTENANCE_HMI_SCREENS_VARIABLES".HMI_SIGNALS.MAINTENANCE_ACTION_LIST_VALUE = 1007);
   "DB17000_MAINTENANCE_GLOBAL_VARIABLES".ACTION_DONE.MACHINE.UNIT_1.GENERAL.PROFILOMETER_LENS_CLEANING := "DB17010_MAINTENANCE_HMI_SCREENS_VARIABLES".HMI_SIGNALS.ACKNOWLEDGE_ACTION_BUTTON AND ("DB17010_MAINTENANCE_HMI_SCREENS_VARIABLES".HMI_SIGNALS.MAINTENANCE_ACTION_LIST_VALUE = 1008);
   "DB17000_MAINTENANCE_GLOBAL_VARIABLES".ACTION_DONE.MACHINE.UNIT_1.GENERAL.PYROMETER_CONFIG_IN_PROGRESS := "DB17010_MAINTENANCE_HMI_SCREENS_VARIABLES".HMI_SIGNALS.ACKNOWLEDGE_ACTION_BUTTON AND ("DB17010_MAINTENANCE_HMI_SCREENS_VARIABLES".HMI_SIGNALS.MAINTENANCE_ACTION_LIST_VALUE = 1009);
   "DB17000_MAINTENANCE_GLOBAL_VARIABLES".ACTION_DONE.MACHINE.UNIT_1.GENERAL.WATER_SYSTEM := "DB17010_MAINTENANCE_HMI_SCREENS_VARIABLES".HMI_SIGNALS.ACKNOWLEDGE_ACTION_BUTTON AND ("DB17010_MAINTENANCE_HMI_SCREENS_VARIABLES".HMI_SIGNALS.MAINTENANCE_ACTION_LIST_VALUE = 1010);
   "DB17000_MAINTENANCE_GLOBAL_VARIABLES".ACTION_DONE.MACHINE.UNIT_1.GENERAL.GAS_SYSTEM := "DB17010_MAINTENANCE_HMI_SCREENS_VARIABLES".HMI_SIGNALS.ACKNOWLEDGE_ACTION_BUTTON AND ("DB17010_MAINTENANCE_HMI_SCREENS_VARIABLES".HMI_SIGNALS.MAINTENANCE_ACTION_LIST_VALUE = 1011);
   "DB17000_MAINTENANCE_GLOBAL_VARIABLES".ACTION_DONE.MACHINE.UNIT_1.GENERAL.AXIS_REFERENCE_SEQUENCE := "DB17010_MAINTENANCE_HMI_SCREENS_VARIABLES".HMI_SIGNALS.ACKNOWLEDGE_ACTION_BUTTON AND ("DB17010_MAINTENANCE_HMI_SCREENS_VARIABLES".HMI_SIGNALS.MAINTENANCE_ACTION_LIST_VALUE = 1012);
   "DB17000_MAINTENANCE_GLOBAL_VARIABLES".ACTION_DONE.MACHINE.UNIT_1.GENERAL.ADJUSTMENT_AXIS_C11 := "DB17010_MAINTENANCE_HMI_SCREENS_VARIABLES".HMI_SIGNALS.ACKNOWLEDGE_ACTION_BUTTON AND ("DB17010_MAINTENANCE_HMI_SCREENS_VARIABLES".HMI_SIGNALS.MAINTENANCE_ACTION_LIST_VALUE = 1013);
   "DB17000_MAINTENANCE_GLOBAL_VARIABLES".ACTION_DONE.MACHINE.UNIT_1.GENERAL.ADJUSTMENT_AXIS_C12 := "DB17010_MAINTENANCE_HMI_SCREENS_VARIABLES".HMI_SIGNALS.ACKNOWLEDGE_ACTION_BUTTON AND ("DB17010_MAINTENANCE_HMI_SCREENS_VARIABLES".HMI_SIGNALS.MAINTENANCE_ACTION_LIST_VALUE = 1014);
   "DB17000_MAINTENANCE_GLOBAL_VARIABLES".ACTION_DONE.MACHINE.UNIT_1.GENERAL.ADJUSTMENT_AXIS_C13 := "DB17010_MAINTENANCE_HMI_SCREENS_VARIABLES".HMI_SIGNALS.ACKNOWLEDGE_ACTION_BUTTON AND ("DB17010_MAINTENANCE_HMI_SCREENS_VARIABLES".HMI_SIGNALS.MAINTENANCE_ACTION_LIST_VALUE = 1015);
   "DB17000_MAINTENANCE_GLOBAL_VARIABLES".ACTION_DONE.MACHINE.UNIT_1.GENERAL.ADJUSTMENT_AXIS_C14 := "DB17010_MAINTENANCE_HMI_SCREENS_VARIABLES".HMI_SIGNALS.ACKNOWLEDGE_ACTION_BUTTON AND ("DB17010_MAINTENANCE_HMI_SCREENS_VARIABLES".HMI_SIGNALS.MAINTENANCE_ACTION_LIST_VALUE = 1016);
   "DB17000_MAINTENANCE_GLOBAL_VARIABLES".ACTION_DONE.MACHINE.UNIT_1.GENERAL.ADJUSTMENT_AXIS_X13 := "DB17010_MAINTENANCE_HMI_SCREENS_VARIABLES".HMI_SIGNALS.ACKNOWLEDGE_ACTION_BUTTON AND ("DB17010_MAINTENANCE_HMI_SCREENS_VARIABLES".HMI_SIGNALS.MAINTENANCE_ACTION_LIST_VALUE = 1017);
   "DB17000_MAINTENANCE_GLOBAL_VARIABLES".ACTION_DONE.MACHINE.UNIT_1.GENERAL.ADJUSTMENT_AXIS_Z13 := "DB17010_MAINTENANCE_HMI_SCREENS_VARIABLES".HMI_SIGNALS.ACKNOWLEDGE_ACTION_BUTTON AND ("DB17010_MAINTENANCE_HMI_SCREENS_VARIABLES".HMI_SIGNALS.MAINTENANCE_ACTION_LIST_VALUE = 1018);
   "DB17000_MAINTENANCE_GLOBAL_VARIABLES".ACTION_DONE.MACHINE.UNIT_1.GENERAL.ADJUSTMENT_AXIS_E10 := "DB17010_MAINTENANCE_HMI_SCREENS_VARIABLES".HMI_SIGNALS.ACKNOWLEDGE_ACTION_BUTTON AND ("DB17010_MAINTENANCE_HMI_SCREENS_VARIABLES".HMI_SIGNALS.MAINTENANCE_ACTION_LIST_VALUE = 1019);
END_REGION

REGION Network 12: ACTION DONE: MACHINE > UNIT 1 > LASER
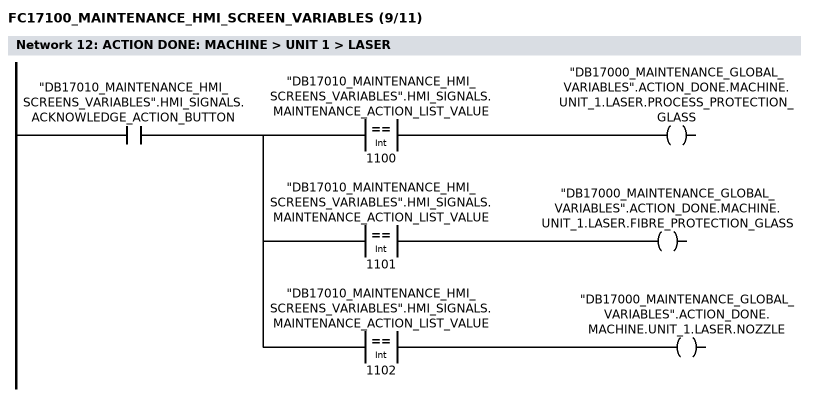
   RUNG wire#powerrail
      Contact( "DB17010_MAINTENANCE_HMI_SCREENS_VARIABLES".HMI_SIGNALS.ACKNOWLEDGE_ACTION_BUTTON )
      wire#w1
      { S7_Templates := "SrcType := Int" } EQ_Contact(in1 := "DB17010_MAINTENANCE_HMI_SCREENS_VARIABLES".HMI_SIGNALS.MAINTENANCE_ACTION_LIST_VALUE, in2 := 1100)
      Coil( "DB17000_MAINTENANCE_GLOBAL_VARIABLES".ACTION_DONE.MACHINE.UNIT_1.LASER.PROCESS_PROTECTION_GLASS )
   END_RUNG
   RUNG wire#w1
      { S7_Templates := "SrcType := Int" } EQ_Contact(in1 := "DB17010_MAINTENANCE_HMI_SCREENS_VARIABLES".HMI_SIGNALS.MAINTENANCE_ACTION_LIST_VALUE, in2 := 1101)
      Coil( "DB17000_MAINTENANCE_GLOBAL_VARIABLES".ACTION_DONE.MACHINE.UNIT_1.LASER.FIBRE_PROTECTION_GLASS )
   END_RUNG
   RUNG wire#w1
      { S7_Templates := "SrcType := Int" } EQ_Contact(in1 := "DB17010_MAINTENANCE_HMI_SCREENS_VARIABLES".HMI_SIGNALS.MAINTENANCE_ACTION_LIST_VALUE, in2 := 1102)
      Coil( "DB17000_MAINTENANCE_GLOBAL_VARIABLES".ACTION_DONE.MACHINE.UNIT_1.LASER.NOZZLE )
   END_RUNG
   // the same network as SCL:
   "DB17000_MAINTENANCE_GLOBAL_VARIABLES".ACTION_DONE.MACHINE.UNIT_1.LASER.PROCESS_PROTECTION_GLASS := "DB17010_MAINTENANCE_HMI_SCREENS_VARIABLES".HMI_SIGNALS.ACKNOWLEDGE_ACTION_BUTTON AND ("DB17010_MAINTENANCE_HMI_SCREENS_VARIABLES".HMI_SIGNALS.MAINTENANCE_ACTION_LIST_VALUE = 1100);
   "DB17000_MAINTENANCE_GLOBAL_VARIABLES".ACTION_DONE.MACHINE.UNIT_1.LASER.FIBRE_PROTECTION_GLASS := "DB17010_MAINTENANCE_HMI_SCREENS_VARIABLES".HMI_SIGNALS.ACKNOWLEDGE_ACTION_BUTTON AND ("DB17010_MAINTENANCE_HMI_SCREENS_VARIABLES".HMI_SIGNALS.MAINTENANCE_ACTION_LIST_VALUE = 1101);
   "DB17000_MAINTENANCE_GLOBAL_VARIABLES".ACTION_DONE.MACHINE.UNIT_1.LASER.NOZZLE := "DB17010_MAINTENANCE_HMI_SCREENS_VARIABLES".HMI_SIGNALS.ACKNOWLEDGE_ACTION_BUTTON AND ("DB17010_MAINTENANCE_HMI_SCREENS_VARIABLES".HMI_SIGNALS.MAINTENANCE_ACTION_LIST_VALUE = 1102);
END_REGION

REGION Network 13: ACTION DONE: MACHINE > UNIT 2 > GENERAL
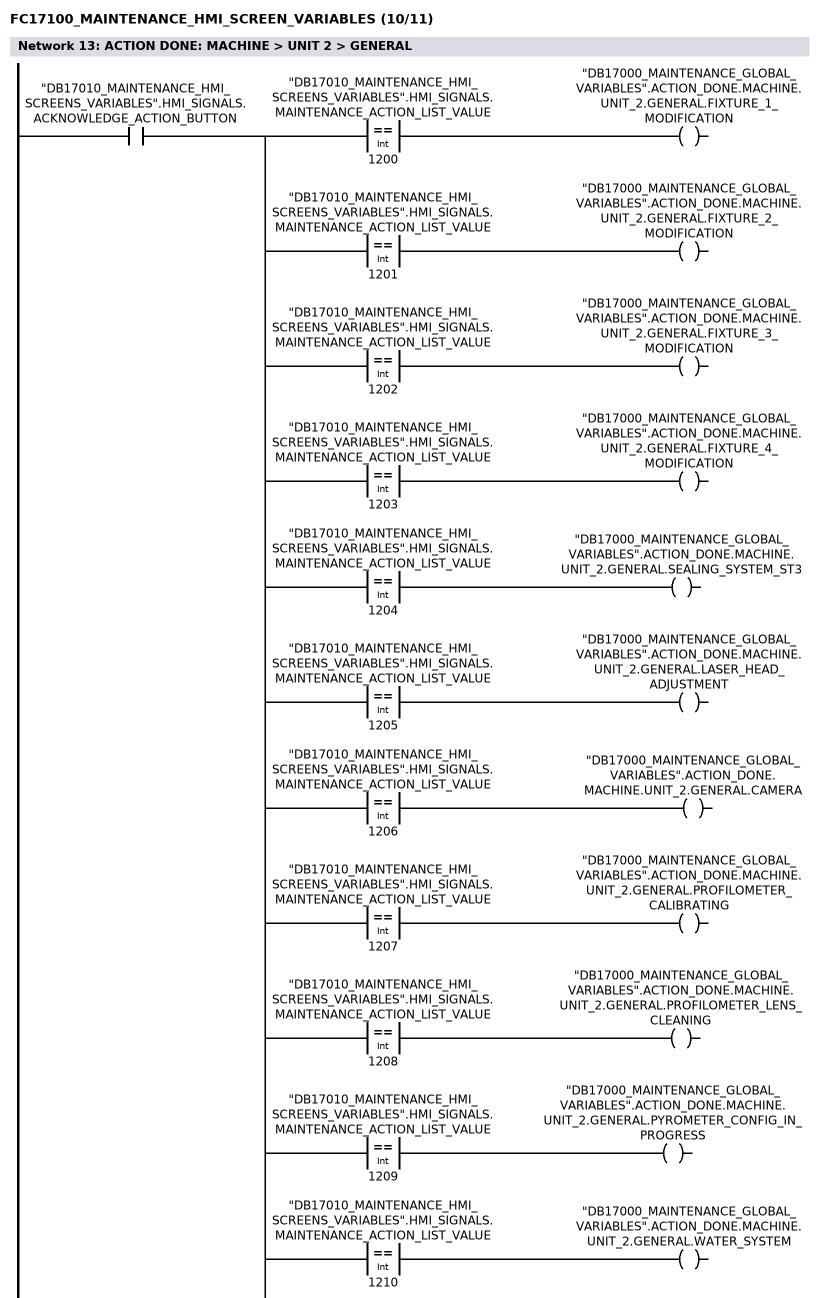
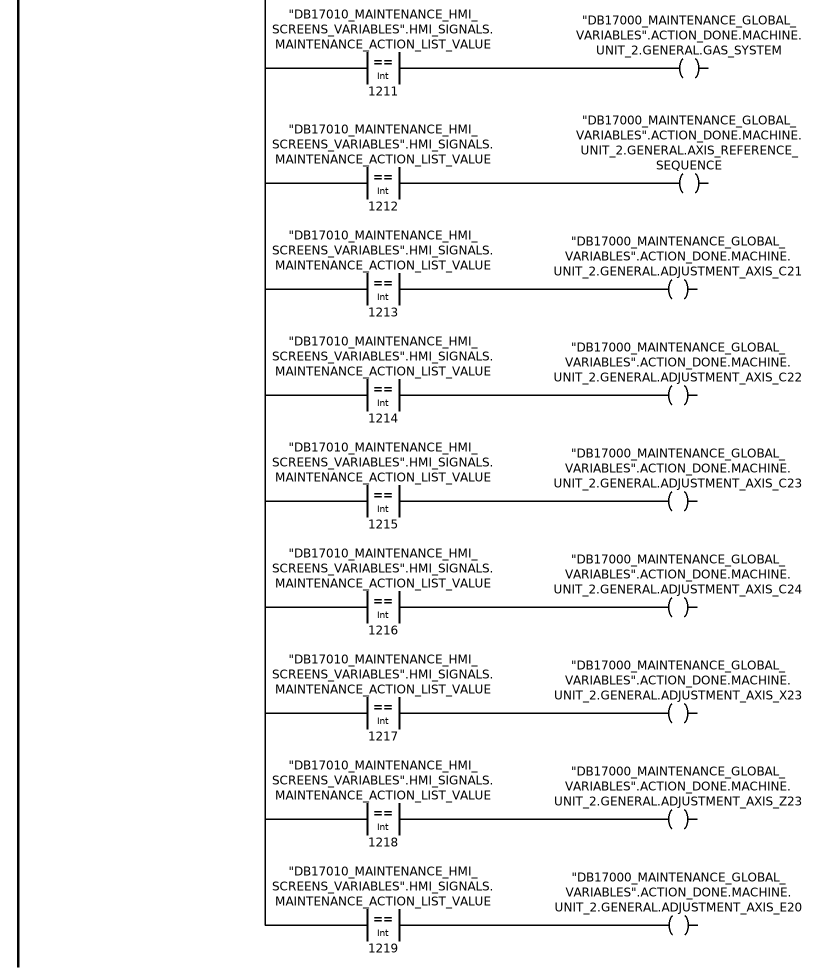
   RUNG wire#powerrail
      Contact( "DB17010_MAINTENANCE_HMI_SCREENS_VARIABLES".HMI_SIGNALS.ACKNOWLEDGE_ACTION_BUTTON )
      wire#w1
      { S7_Templates := "SrcType := Int" } EQ_Contact(in1 := "DB17010_MAINTENANCE_HMI_SCREENS_VARIABLES".HMI_SIGNALS.MAINTENANCE_ACTION_LIST_VALUE, in2 := 1200)
      Coil( "DB17000_MAINTENANCE_GLOBAL_VARIABLES".ACTION_DONE.MACHINE.UNIT_2.GENERAL.FIXTURE_1_MODIFICATION )
   END_RUNG
   RUNG wire#w1
      { S7_Templates := "SrcType := Int" } EQ_Contact(in1 := "DB17010_MAINTENANCE_HMI_SCREENS_VARIABLES".HMI_SIGNALS.MAINTENANCE_ACTION_LIST_VALUE, in2 := 1201)
      Coil( "DB17000_MAINTENANCE_GLOBAL_VARIABLES".ACTION_DONE.MACHINE.UNIT_2.GENERAL.FIXTURE_2_MODIFICATION )
   END_RUNG
   RUNG wire#w1
      { S7_Templates := "SrcType := Int" } EQ_Contact(in1 := "DB17010_MAINTENANCE_HMI_SCREENS_VARIABLES".HMI_SIGNALS.MAINTENANCE_ACTION_LIST_VALUE, in2 := 1202)
      Coil( "DB17000_MAINTENANCE_GLOBAL_VARIABLES".ACTION_DONE.MACHINE.UNIT_2.GENERAL.FIXTURE_3_MODIFICATION )
   END_RUNG
   RUNG wire#w1
      { S7_Templates := "SrcType := Int" } EQ_Contact(in1 := "DB17010_MAINTENANCE_HMI_SCREENS_VARIABLES".HMI_SIGNALS.MAINTENANCE_ACTION_LIST_VALUE, in2 := 1203)
      Coil( "DB17000_MAINTENANCE_GLOBAL_VARIABLES".ACTION_DONE.MACHINE.UNIT_2.GENERAL.FIXTURE_4_MODIFICATION )
   END_RUNG
   RUNG wire#w1
      { S7_Templates := "SrcType := Int" } EQ_Contact(in1 := "DB17010_MAINTENANCE_HMI_SCREENS_VARIABLES".HMI_SIGNALS.MAINTENANCE_ACTION_LIST_VALUE, in2 := 1204)
      Coil( "DB17000_MAINTENANCE_GLOBAL_VARIABLES".ACTION_DONE.MACHINE.UNIT_2.GENERAL.SEALING_SYSTEM_ST3 )
   END_RUNG
   RUNG wire#w1
      { S7_Templates := "SrcType := Int" } EQ_Contact(in1 := "DB17010_MAINTENANCE_HMI_SCREENS_VARIABLES".HMI_SIGNALS.MAINTENANCE_ACTION_LIST_VALUE, in2 := 1205)
      Coil( "DB17000_MAINTENANCE_GLOBAL_VARIABLES".ACTION_DONE.MACHINE.UNIT_2.GENERAL.LASER_HEAD_ADJUSTMENT )
   END_RUNG
   RUNG wire#w1
      { S7_Templates := "SrcType := Int" } EQ_Contact(in1 := "DB17010_MAINTENANCE_HMI_SCREENS_VARIABLES".HMI_SIGNALS.MAINTENANCE_ACTION_LIST_VALUE, in2 := 1206)
      Coil( "DB17000_MAINTENANCE_GLOBAL_VARIABLES".ACTION_DONE.MACHINE.UNIT_2.GENERAL.CAMERA )
   END_RUNG
   RUNG wire#w1
      { S7_Templates := "SrcType := Int" } EQ_Contact(in1 := "DB17010_MAINTENANCE_HMI_SCREENS_VARIABLES".HMI_SIGNALS.MAINTENANCE_ACTION_LIST_VALUE, in2 := 1207)
      Coil( "DB17000_MAINTENANCE_GLOBAL_VARIABLES".ACTION_DONE.MACHINE.UNIT_2.GENERAL.PROFILOMETER_CALIBRATING )
   END_RUNG
   RUNG wire#w1
      { S7_Templates := "SrcType := Int" } EQ_Contact(in1 := "DB17010_MAINTENANCE_HMI_SCREENS_VARIABLES".HMI_SIGNALS.MAINTENANCE_ACTION_LIST_VALUE, in2 := 1208)
      Coil( "DB17000_MAINTENANCE_GLOBAL_VARIABLES".ACTION_DONE.MACHINE.UNIT_2.GENERAL.PROFILOMETER_LENS_CLEANING )
   END_RUNG
   RUNG wire#w1
      { S7_Templates := "SrcType := Int" } EQ_Contact(in1 := "DB17010_MAINTENANCE_HMI_SCREENS_VARIABLES".HMI_SIGNALS.MAINTENANCE_ACTION_LIST_VALUE, in2 := 1209)
      Coil( "DB17000_MAINTENANCE_GLOBAL_VARIABLES".ACTION_DONE.MACHINE.UNIT_2.GENERAL.PYROMETER_CONFIG_IN_PROGRESS )
   END_RUNG
   RUNG wire#w1
      { S7_Templates := "SrcType := Int" } EQ_Contact(in1 := "DB17010_MAINTENANCE_HMI_SCREENS_VARIABLES".HMI_SIGNALS.MAINTENANCE_ACTION_LIST_VALUE, in2 := 1210)
      Coil( "DB17000_MAINTENANCE_GLOBAL_VARIABLES".ACTION_DONE.MACHINE.UNIT_2.GENERAL.WATER_SYSTEM )
   END_RUNG
   RUNG wire#w1
      { S7_Templates := "SrcType := Int" } EQ_Contact(in1 := "DB17010_MAINTENANCE_HMI_SCREENS_VARIABLES".HMI_SIGNALS.MAINTENANCE_ACTION_LIST_VALUE, in2 := 1211)
      Coil( "DB17000_MAINTENANCE_GLOBAL_VARIABLES".ACTION_DONE.MACHINE.UNIT_2.GENERAL.GAS_SYSTEM )
   END_RUNG
   RUNG wire#w1
      { S7_Templates := "SrcType := Int" } EQ_Contact(in1 := "DB17010_MAINTENANCE_HMI_SCREENS_VARIABLES".HMI_SIGNALS.MAINTENANCE_ACTION_LIST_VALUE, in2 := 1212)
      Coil( "DB17000_MAINTENANCE_GLOBAL_VARIABLES".ACTION_DONE.MACHINE.UNIT_2.GENERAL.AXIS_REFERENCE_SEQUENCE )
   END_RUNG
   RUNG wire#w1
      { S7_Templates := "SrcType := Int" } EQ_Contact(in1 := "DB17010_MAINTENANCE_HMI_SCREENS_VARIABLES".HMI_SIGNALS.MAINTENANCE_ACTION_LIST_VALUE, in2 := 1213)
      Coil( "DB17000_MAINTENANCE_GLOBAL_VARIABLES".ACTION_DONE.MACHINE.UNIT_2.GENERAL.ADJUSTMENT_AXIS_C21 )
   END_RUNG
   RUNG wire#w1
      { S7_Templates := "SrcType := Int" } EQ_Contact(in1 := "DB17010_MAINTENANCE_HMI_SCREENS_VARIABLES".HMI_SIGNALS.MAINTENANCE_ACTION_LIST_VALUE, in2 := 1214)
      Coil( "DB17000_MAINTENANCE_GLOBAL_VARIABLES".ACTION_DONE.MACHINE.UNIT_2.GENERAL.ADJUSTMENT_AXIS_C22 )
   END_RUNG
   RUNG wire#w1
      { S7_Templates := "SrcType := Int" } EQ_Contact(in1 := "DB17010_MAINTENANCE_HMI_SCREENS_VARIABLES".HMI_SIGNALS.MAINTENANCE_ACTION_LIST_VALUE, in2 := 1215)
      Coil( "DB17000_MAINTENANCE_GLOBAL_VARIABLES".ACTION_DONE.MACHINE.UNIT_2.GENERAL.ADJUSTMENT_AXIS_C23 )
   END_RUNG
   RUNG wire#w1
      { S7_Templates := "SrcType := Int" } EQ_Contact(in1 := "DB17010_MAINTENANCE_HMI_SCREENS_VARIABLES".HMI_SIGNALS.MAINTENANCE_ACTION_LIST_VALUE, in2 := 1216)
      Coil( "DB17000_MAINTENANCE_GLOBAL_VARIABLES".ACTION_DONE.MACHINE.UNIT_2.GENERAL.ADJUSTMENT_AXIS_C24 )
   END_RUNG
   RUNG wire#w1
      { S7_Templates := "SrcType := Int" } EQ_Contact(in1 := "DB17010_MAINTENANCE_HMI_SCREENS_VARIABLES".HMI_SIGNALS.MAINTENANCE_ACTION_LIST_VALUE, in2 := 1217)
      Coil( "DB17000_MAINTENANCE_GLOBAL_VARIABLES".ACTION_DONE.MACHINE.UNIT_2.GENERAL.ADJUSTMENT_AXIS_X23 )
   END_RUNG
   RUNG wire#w1
      { S7_Templates := "SrcType := Int" } EQ_Contact(in1 := "DB17010_MAINTENANCE_HMI_SCREENS_VARIABLES".HMI_SIGNALS.MAINTENANCE_ACTION_LIST_VALUE, in2 := 1218)
      Coil( "DB17000_MAINTENANCE_GLOBAL_VARIABLES".ACTION_DONE.MACHINE.UNIT_2.GENERAL.ADJUSTMENT_AXIS_Z23 )
   END_RUNG
   RUNG wire#w1
      { S7_Templates := "SrcType := Int" } EQ_Contact(in1 := "DB17010_MAINTENANCE_HMI_SCREENS_VARIABLES".HMI_SIGNALS.MAINTENANCE_ACTION_LIST_VALUE, in2 := 1219)
      Coil( "DB17000_MAINTENANCE_GLOBAL_VARIABLES".ACTION_DONE.MACHINE.UNIT_2.GENERAL.ADJUSTMENT_AXIS_E20 )
   END_RUNG
   // the same network as SCL:
   "DB17000_MAINTENANCE_GLOBAL_VARIABLES".ACTION_DONE.MACHINE.UNIT_2.GENERAL.FIXTURE_1_MODIFICATION := "DB17010_MAINTENANCE_HMI_SCREENS_VARIABLES".HMI_SIGNALS.ACKNOWLEDGE_ACTION_BUTTON AND ("DB17010_MAINTENANCE_HMI_SCREENS_VARIABLES".HMI_SIGNALS.MAINTENANCE_ACTION_LIST_VALUE = 1200);
   "DB17000_MAINTENANCE_GLOBAL_VARIABLES".ACTION_DONE.MACHINE.UNIT_2.GENERAL.FIXTURE_2_MODIFICATION := "DB17010_MAINTENANCE_HMI_SCREENS_VARIABLES".HMI_SIGNALS.ACKNOWLEDGE_ACTION_BUTTON AND ("DB17010_MAINTENANCE_HMI_SCREENS_VARIABLES".HMI_SIGNALS.MAINTENANCE_ACTION_LIST_VALUE = 1201);
   "DB17000_MAINTENANCE_GLOBAL_VARIABLES".ACTION_DONE.MACHINE.UNIT_2.GENERAL.FIXTURE_3_MODIFICATION := "DB17010_MAINTENANCE_HMI_SCREENS_VARIABLES".HMI_SIGNALS.ACKNOWLEDGE_ACTION_BUTTON AND ("DB17010_MAINTENANCE_HMI_SCREENS_VARIABLES".HMI_SIGNALS.MAINTENANCE_ACTION_LIST_VALUE = 1202);
   "DB17000_MAINTENANCE_GLOBAL_VARIABLES".ACTION_DONE.MACHINE.UNIT_2.GENERAL.FIXTURE_4_MODIFICATION := "DB17010_MAINTENANCE_HMI_SCREENS_VARIABLES".HMI_SIGNALS.ACKNOWLEDGE_ACTION_BUTTON AND ("DB17010_MAINTENANCE_HMI_SCREENS_VARIABLES".HMI_SIGNALS.MAINTENANCE_ACTION_LIST_VALUE = 1203);
   "DB17000_MAINTENANCE_GLOBAL_VARIABLES".ACTION_DONE.MACHINE.UNIT_2.GENERAL.SEALING_SYSTEM_ST3 := "DB17010_MAINTENANCE_HMI_SCREENS_VARIABLES".HMI_SIGNALS.ACKNOWLEDGE_ACTION_BUTTON AND ("DB17010_MAINTENANCE_HMI_SCREENS_VARIABLES".HMI_SIGNALS.MAINTENANCE_ACTION_LIST_VALUE = 1204);
   "DB17000_MAINTENANCE_GLOBAL_VARIABLES".ACTION_DONE.MACHINE.UNIT_2.GENERAL.LASER_HEAD_ADJUSTMENT := "DB17010_MAINTENANCE_HMI_SCREENS_VARIABLES".HMI_SIGNALS.ACKNOWLEDGE_ACTION_BUTTON AND ("DB17010_MAINTENANCE_HMI_SCREENS_VARIABLES".HMI_SIGNALS.MAINTENANCE_ACTION_LIST_VALUE = 1205);
   "DB17000_MAINTENANCE_GLOBAL_VARIABLES".ACTION_DONE.MACHINE.UNIT_2.GENERAL.CAMERA := "DB17010_MAINTENANCE_HMI_SCREENS_VARIABLES".HMI_SIGNALS.ACKNOWLEDGE_ACTION_BUTTON AND ("DB17010_MAINTENANCE_HMI_SCREENS_VARIABLES".HMI_SIGNALS.MAINTENANCE_ACTION_LIST_VALUE = 1206);
   "DB17000_MAINTENANCE_GLOBAL_VARIABLES".ACTION_DONE.MACHINE.UNIT_2.GENERAL.PROFILOMETER_CALIBRATING := "DB17010_MAINTENANCE_HMI_SCREENS_VARIABLES".HMI_SIGNALS.ACKNOWLEDGE_ACTION_BUTTON AND ("DB17010_MAINTENANCE_HMI_SCREENS_VARIABLES".HMI_SIGNALS.MAINTENANCE_ACTION_LIST_VALUE = 1207);
   "DB17000_MAINTENANCE_GLOBAL_VARIABLES".ACTION_DONE.MACHINE.UNIT_2.GENERAL.PROFILOMETER_LENS_CLEANING := "DB17010_MAINTENANCE_HMI_SCREENS_VARIABLES".HMI_SIGNALS.ACKNOWLEDGE_ACTION_BUTTON AND ("DB17010_MAINTENANCE_HMI_SCREENS_VARIABLES".HMI_SIGNALS.MAINTENANCE_ACTION_LIST_VALUE = 1208);
   "DB17000_MAINTENANCE_GLOBAL_VARIABLES".ACTION_DONE.MACHINE.UNIT_2.GENERAL.PYROMETER_CONFIG_IN_PROGRESS := "DB17010_MAINTENANCE_HMI_SCREENS_VARIABLES".HMI_SIGNALS.ACKNOWLEDGE_ACTION_BUTTON AND ("DB17010_MAINTENANCE_HMI_SCREENS_VARIABLES".HMI_SIGNALS.MAINTENANCE_ACTION_LIST_VALUE = 1209);
   "DB17000_MAINTENANCE_GLOBAL_VARIABLES".ACTION_DONE.MACHINE.UNIT_2.GENERAL.WATER_SYSTEM := "DB17010_MAINTENANCE_HMI_SCREENS_VARIABLES".HMI_SIGNALS.ACKNOWLEDGE_ACTION_BUTTON AND ("DB17010_MAINTENANCE_HMI_SCREENS_VARIABLES".HMI_SIGNALS.MAINTENANCE_ACTION_LIST_VALUE = 1210);
   "DB17000_MAINTENANCE_GLOBAL_VARIABLES".ACTION_DONE.MACHINE.UNIT_2.GENERAL.GAS_SYSTEM := "DB17010_MAINTENANCE_HMI_SCREENS_VARIABLES".HMI_SIGNALS.ACKNOWLEDGE_ACTION_BUTTON AND ("DB17010_MAINTENANCE_HMI_SCREENS_VARIABLES".HMI_SIGNALS.MAINTENANCE_ACTION_LIST_VALUE = 1211);
   "DB17000_MAINTENANCE_GLOBAL_VARIABLES".ACTION_DONE.MACHINE.UNIT_2.GENERAL.AXIS_REFERENCE_SEQUENCE := "DB17010_MAINTENANCE_HMI_SCREENS_VARIABLES".HMI_SIGNALS.ACKNOWLEDGE_ACTION_BUTTON AND ("DB17010_MAINTENANCE_HMI_SCREENS_VARIABLES".HMI_SIGNALS.MAINTENANCE_ACTION_LIST_VALUE = 1212);
   "DB17000_MAINTENANCE_GLOBAL_VARIABLES".ACTION_DONE.MACHINE.UNIT_2.GENERAL.ADJUSTMENT_AXIS_C21 := "DB17010_MAINTENANCE_HMI_SCREENS_VARIABLES".HMI_SIGNALS.ACKNOWLEDGE_ACTION_BUTTON AND ("DB17010_MAINTENANCE_HMI_SCREENS_VARIABLES".HMI_SIGNALS.MAINTENANCE_ACTION_LIST_VALUE = 1213);
   "DB17000_MAINTENANCE_GLOBAL_VARIABLES".ACTION_DONE.MACHINE.UNIT_2.GENERAL.ADJUSTMENT_AXIS_C22 := "DB17010_MAINTENANCE_HMI_SCREENS_VARIABLES".HMI_SIGNALS.ACKNOWLEDGE_ACTION_BUTTON AND ("DB17010_MAINTENANCE_HMI_SCREENS_VARIABLES".HMI_SIGNALS.MAINTENANCE_ACTION_LIST_VALUE = 1214);
   "DB17000_MAINTENANCE_GLOBAL_VARIABLES".ACTION_DONE.MACHINE.UNIT_2.GENERAL.ADJUSTMENT_AXIS_C23 := "DB17010_MAINTENANCE_HMI_SCREENS_VARIABLES".HMI_SIGNALS.ACKNOWLEDGE_ACTION_BUTTON AND ("DB17010_MAINTENANCE_HMI_SCREENS_VARIABLES".HMI_SIGNALS.MAINTENANCE_ACTION_LIST_VALUE = 1215);
   "DB17000_MAINTENANCE_GLOBAL_VARIABLES".ACTION_DONE.MACHINE.UNIT_2.GENERAL.ADJUSTMENT_AXIS_C24 := "DB17010_MAINTENANCE_HMI_SCREENS_VARIABLES".HMI_SIGNALS.ACKNOWLEDGE_ACTION_BUTTON AND ("DB17010_MAINTENANCE_HMI_SCREENS_VARIABLES".HMI_SIGNALS.MAINTENANCE_ACTION_LIST_VALUE = 1216);
   "DB17000_MAINTENANCE_GLOBAL_VARIABLES".ACTION_DONE.MACHINE.UNIT_2.GENERAL.ADJUSTMENT_AXIS_X23 := "DB17010_MAINTENANCE_HMI_SCREENS_VARIABLES".HMI_SIGNALS.ACKNOWLEDGE_ACTION_BUTTON AND ("DB17010_MAINTENANCE_HMI_SCREENS_VARIABLES".HMI_SIGNALS.MAINTENANCE_ACTION_LIST_VALUE = 1217);
   "DB17000_MAINTENANCE_GLOBAL_VARIABLES".ACTION_DONE.MACHINE.UNIT_2.GENERAL.ADJUSTMENT_AXIS_Z23 := "DB17010_MAINTENANCE_HMI_SCREENS_VARIABLES".HMI_SIGNALS.ACKNOWLEDGE_ACTION_BUTTON AND ("DB17010_MAINTENANCE_HMI_SCREENS_VARIABLES".HMI_SIGNALS.MAINTENANCE_ACTION_LIST_VALUE = 1218);
   "DB17000_MAINTENANCE_GLOBAL_VARIABLES".ACTION_DONE.MACHINE.UNIT_2.GENERAL.ADJUSTMENT_AXIS_E20 := "DB17010_MAINTENANCE_HMI_SCREENS_VARIABLES".HMI_SIGNALS.ACKNOWLEDGE_ACTION_BUTTON AND ("DB17010_MAINTENANCE_HMI_SCREENS_VARIABLES".HMI_SIGNALS.MAINTENANCE_ACTION_LIST_VALUE = 1219);
END_REGION

REGION Network 14: ACTION DONE: MACHINE > UNIT 2 > LASER
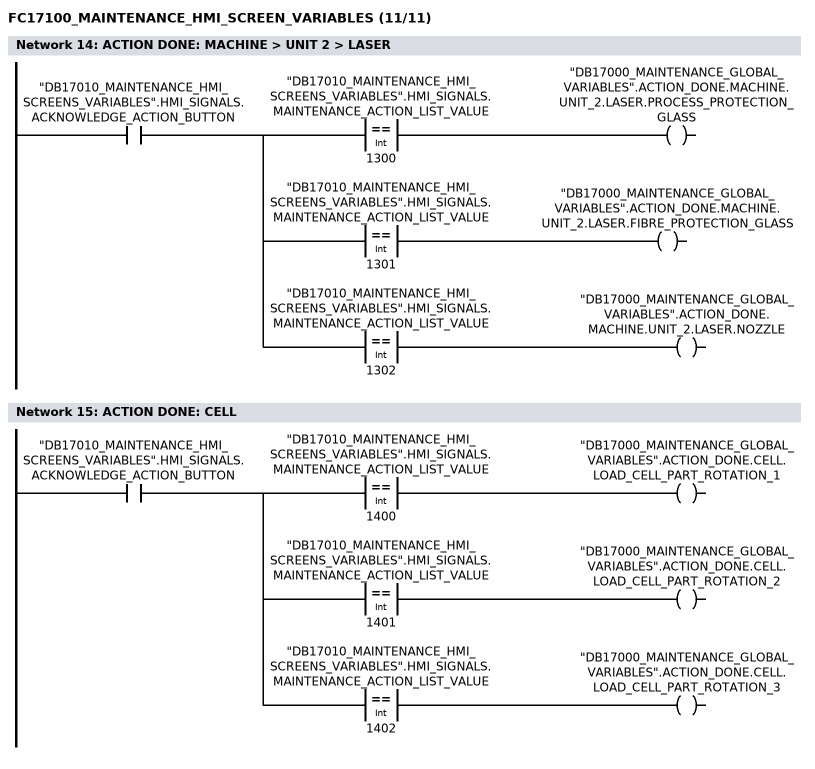
   RUNG wire#powerrail
      Contact( "DB17010_MAINTENANCE_HMI_SCREENS_VARIABLES".HMI_SIGNALS.ACKNOWLEDGE_ACTION_BUTTON )
      wire#w1
      { S7_Templates := "SrcType := Int" } EQ_Contact(in1 := "DB17010_MAINTENANCE_HMI_SCREENS_VARIABLES".HMI_SIGNALS.MAINTENANCE_ACTION_LIST_VALUE, in2 := 1300)
      Coil( "DB17000_MAINTENANCE_GLOBAL_VARIABLES".ACTION_DONE.MACHINE.UNIT_2.LASER.PROCESS_PROTECTION_GLASS )
   END_RUNG
   RUNG wire#w1
      { S7_Templates := "SrcType := Int" } EQ_Contact(in1 := "DB17010_MAINTENANCE_HMI_SCREENS_VARIABLES".HMI_SIGNALS.MAINTENANCE_ACTION_LIST_VALUE, in2 := 1301)
      Coil( "DB17000_MAINTENANCE_GLOBAL_VARIABLES".ACTION_DONE.MACHINE.UNIT_2.LASER.FIBRE_PROTECTION_GLASS )
   END_RUNG
   RUNG wire#w1
      { S7_Templates := "SrcType := Int" } EQ_Contact(in1 := "DB17010_MAINTENANCE_HMI_SCREENS_VARIABLES".HMI_SIGNALS.MAINTENANCE_ACTION_LIST_VALUE, in2 := 1302)
      Coil( "DB17000_MAINTENANCE_GLOBAL_VARIABLES".ACTION_DONE.MACHINE.UNIT_2.LASER.NOZZLE )
   END_RUNG
   // the same network as SCL:
   "DB17000_MAINTENANCE_GLOBAL_VARIABLES".ACTION_DONE.MACHINE.UNIT_2.LASER.PROCESS_PROTECTION_GLASS := "DB17010_MAINTENANCE_HMI_SCREENS_VARIABLES".HMI_SIGNALS.ACKNOWLEDGE_ACTION_BUTTON AND ("DB17010_MAINTENANCE_HMI_SCREENS_VARIABLES".HMI_SIGNALS.MAINTENANCE_ACTION_LIST_VALUE = 1300);
   "DB17000_MAINTENANCE_GLOBAL_VARIABLES".ACTION_DONE.MACHINE.UNIT_2.LASER.FIBRE_PROTECTION_GLASS := "DB17010_MAINTENANCE_HMI_SCREENS_VARIABLES".HMI_SIGNALS.ACKNOWLEDGE_ACTION_BUTTON AND ("DB17010_MAINTENANCE_HMI_SCREENS_VARIABLES".HMI_SIGNALS.MAINTENANCE_ACTION_LIST_VALUE = 1301);
   "DB17000_MAINTENANCE_GLOBAL_VARIABLES".ACTION_DONE.MACHINE.UNIT_2.LASER.NOZZLE := "DB17010_MAINTENANCE_HMI_SCREENS_VARIABLES".HMI_SIGNALS.ACKNOWLEDGE_ACTION_BUTTON AND ("DB17010_MAINTENANCE_HMI_SCREENS_VARIABLES".HMI_SIGNALS.MAINTENANCE_ACTION_LIST_VALUE = 1302);
END_REGION

REGION Network 15: ACTION DONE: CELL
   RUNG wire#powerrail
      Contact( "DB17010_MAINTENANCE_HMI_SCREENS_VARIABLES".HMI_SIGNALS.ACKNOWLEDGE_ACTION_BUTTON )
      wire#w1
      { S7_Templates := "SrcType := Int" } EQ_Contact(in1 := "DB17010_MAINTENANCE_HMI_SCREENS_VARIABLES".HMI_SIGNALS.MAINTENANCE_ACTION_LIST_VALUE, in2 := 1400)
      Coil( "DB17000_MAINTENANCE_GLOBAL_VARIABLES".ACTION_DONE.CELL.LOAD_CELL_PART_ROTATION_1 )
   END_RUNG
   RUNG wire#w1
      { S7_Templates := "SrcType := Int" } EQ_Contact(in1 := "DB17010_MAINTENANCE_HMI_SCREENS_VARIABLES".HMI_SIGNALS.MAINTENANCE_ACTION_LIST_VALUE, in2 := 1401)
      Coil( "DB17000_MAINTENANCE_GLOBAL_VARIABLES".ACTION_DONE.CELL.LOAD_CELL_PART_ROTATION_2 )
   END_RUNG
   RUNG wire#w1
      { S7_Templates := "SrcType := Int" } EQ_Contact(in1 := "DB17010_MAINTENANCE_HMI_SCREENS_VARIABLES".HMI_SIGNALS.MAINTENANCE_ACTION_LIST_VALUE, in2 := 1402)
      Coil( "DB17000_MAINTENANCE_GLOBAL_VARIABLES".ACTION_DONE.CELL.LOAD_CELL_PART_ROTATION_3 )
   END_RUNG
   // the same network as SCL:
   "DB17000_MAINTENANCE_GLOBAL_VARIABLES".ACTION_DONE.CELL.LOAD_CELL_PART_ROTATION_1 := "DB17010_MAINTENANCE_HMI_SCREENS_VARIABLES".HMI_SIGNALS.ACKNOWLEDGE_ACTION_BUTTON AND ("DB17010_MAINTENANCE_HMI_SCREENS_VARIABLES".HMI_SIGNALS.MAINTENANCE_ACTION_LIST_VALUE = 1400);
   "DB17000_MAINTENANCE_GLOBAL_VARIABLES".ACTION_DONE.CELL.LOAD_CELL_PART_ROTATION_2 := "DB17010_MAINTENANCE_HMI_SCREENS_VARIABLES".HMI_SIGNALS.ACKNOWLEDGE_ACTION_BUTTON AND ("DB17010_MAINTENANCE_HMI_SCREENS_VARIABLES".HMI_SIGNALS.MAINTENANCE_ACTION_LIST_VALUE = 1401);
   "DB17000_MAINTENANCE_GLOBAL_VARIABLES".ACTION_DONE.CELL.LOAD_CELL_PART_ROTATION_3 := "DB17010_MAINTENANCE_HMI_SCREENS_VARIABLES".HMI_SIGNALS.ACKNOWLEDGE_ACTION_BUTTON AND ("DB17010_MAINTENANCE_HMI_SCREENS_VARIABLES".HMI_SIGNALS.MAINTENANCE_ACTION_LIST_VALUE = 1402);
END_REGION

REGION Network 16 (SCL): OPERATOR HELP
   #NUM_OF_HELPS_TO_0 := 0;
   FOR #TEMP := 0 TO 100 DO
       IF "DB17100_MAINTENANCE_OPERATOR_HELP".OPERATOR_HELP[#TEMP] = 1 THEN
           "DB17010_MAINTENANCE_HMI_SCREENS_VARIABLES".HMI_SIGNALS.OPERATOR_HELP_VALUE := #TEMP;
       ELSE
           #NUM_OF_HELPS_TO_0 := #NUM_OF_HELPS_TO_0 + 1; //Counts number of operator helps that are switched off
       END_IF;
   END_FOR;

   IF #NUM_OF_HELPS_TO_0 = 101 THEN //If all the operator helps are switched off operator help value is set to 0 value
       "DB17010_MAINTENANCE_HMI_SCREENS_VARIABLES".HMI_SIGNALS.OPERATOR_HELP_VALUE := 0;
   END_IF;
END_REGION
END_FUNCTION
